KUKA KRL program: MyProgram_291().src

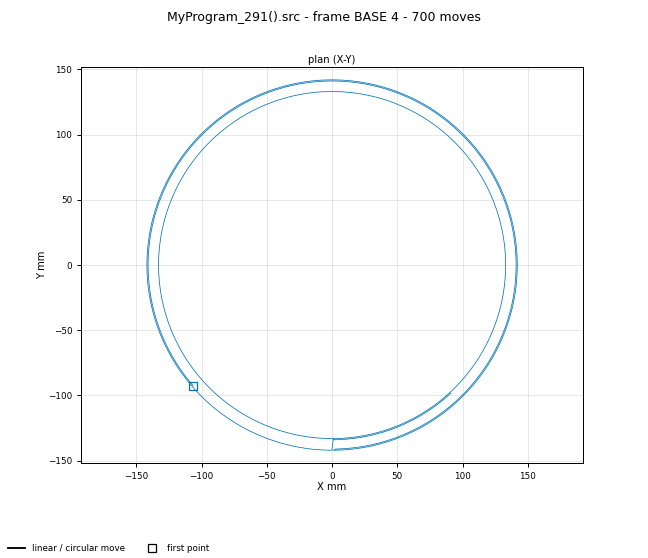
[picture p0: tool path of MyProgram_291().src in frame BASE 4, 700 of 700 moves have a stored position in this frame; points joined in program order, loops and branches not executed]
&ACCESS RVP
&REL 1
&PARAM TEMPLATE = C:\KRC\Roboter\Template\vorgabe
&PARAM EDITMASK = *
DEF MyProgram_291()
; ---- Setting reference (Base) ----
$BASE = BASE_DATA[4]

; --------------------------
; ---- Setting tool (TCP) ----
$TOOL = TOOL_DATA[3]
; --------------------------

$VEL.CP = VEL_APROX_PRINT
Startdeposition()
$VEL.CP = VEL_PRINT
LIN {X -106.5976,Y -92.4172,Z 176,A -136.4755,B 6.9518,C 0.3757,E1 6.8407,E2 228.6931} C_DIS
LIN {X -109.4772,Y -88.9868,Z 176,A -138.3075,B 6.952,C 0.3719,E1 6.8374,E2 230.5261} C_DIS
LIN {X -112.3182,Y -85.3731,Z 176,A -140.1975,B 6.9522,C 0.3681,E1 6.8342,E2 232.4184} C_DIS
LIN {X -114.9882,Y -81.7412,Z 176,A -142.0435,B 6.9524,C 0.3642,E1 6.8312,E2 234.2657} C_DIS
LIN {X -117.5398,Y -78.0276,Z 176,A -143.785,B 6.9527,C 0.3587,E1 6.8285,E2 235.9948} C_DIS
LIN {X -119.6611,Y -74.7331,Z 176,A -145.5405,B 6.9527,C 0.3571,E1 6.8258,E2 237.771} C_DIS
LIN {X -122.1664,Y -70.5632,Z 176,A -148.2334,B 6.9525,C 0.3616,E1 6.8219,E2 240.5556} C_DIS
LIN {X -125.0381,Y -65.3358,Z 176,A -149.8985,B 6.9533,C 0.3458,E1 6.8199,E2 242.1216} C_DIS
LIN {X -126.4778,Y -62.5025,Z 176,A -151.2741,B 6.9534,C 0.3436,E1 6.8181,E2 243.5075} C_DIS
LIN {X -128.0398,Y -59.237,Z 176,A -152.7086,B 6.9536,C 0.3394,E1 6.8164,E2 244.9366} C_DIS
LIN {X -129.8391,Y -55.1885,Z 176,A -154.746,B 6.9537,C 0.3378,E1 6.8141,E2 247.0039} C_DIS
LIN {X -131.2968,Y -51.6206,Z 176,A -156.1181,B 6.954,C 0.3312,E1 6.8127,E2 248.35} C_DIS
LIN {X -132.5485,Y -48.3154,Z 176,A -157.6493,B 6.9541,C 0.3286,E1 6.8112,E2 249.8927} C_DIS
LIN {X -133.6813,Y -45.0871,Z 176,A -158.9184,B 6.9544,C 0.3233,E1 6.8101,E2 251.1454} C_DIS
LIN {X -134.8654,Y -41.4075,Z 176,A -160.6121,B 6.9545,C 0.3207,E1 6.8086,E2 252.854} C_DIS
LIN {X -135.8285,Y -38.13,Z 176,A -162.047,B 6.9547,C 0.3175,E1 6.8075,E2 254.2942} C_DIS
LIN {X -136.7359,Y -34.7357,Z 176,A -163.3925,B 6.9549,C 0.3125,E1 6.8066,E2 255.628} C_DIS
LIN {X -137.4207,Y -31.9236,Z 176,A -164.649,B 6.9549,C 0.3103,E1 6.8058,E2 256.8943} C_DIS
LIN {X -138.1072,Y -28.8125,Z 176,A -165.9668,B 6.9551,C 0.307,E1 6.805,E2 258.2142} C_DIS
LIN {X -138.843,Y -25.0187,Z 176,A -167.6355,B 6.9553,C 0.3038,E1 6.8041,E2 259.8946} C_DIS
LIN {X -139.8868,Y -18.3035,Z 176,A -170.3898,B 6.9556,C 0.2959,E1 6.803,E2 262.6461} C_DIS
LIN {X -140.6363,Y -11.191,Z 176,A -173.5234,B 6.9558,C 0.2905,E1 6.8021,E2 265.8071} C_DIS
LIN {X -140.8895,Y -7.3194,Z 176,A -175.0544,B 6.956,C 0.2855,E1 6.8018,E2 267.3309} C_DIS
LIN {X -141.0677,Y -1.8699,Z 176,A -177.6099,B 6.9561,C 0.2833,E1 6.8017,E2 269.9283} C_DIS
LIN {X -141.0709,Y 1.6738,Z 176,A -178.7902,B 6.9564,C 0.276,E1 6.8017,E2 271.0743} C_DIS
LIN {X -140.9646,Y 5.6916,Z 176,A 179.5595,B 6.9566,C 0.2715,E1 6.8019,E2 272.7255} C_DIS
LIN {X -140.7276,Y 9.9587,Z 176,A 177.6568,B 6.9567,C 0.2686,E1 6.8022,E2 274.6481} C_DIS
LIN {X -139.9779,Y 17.6081,Z 176,A 174.5631,B 6.9571,C 0.2594,E1 6.8031,E2 277.7356} C_DIS
LIN {X -139.1333,Y 23.3505,Z 176,A 172.4063,B 6.9574,C 0.2502,E1 6.804,E2 279.8646} C_DIS
LIN {X -138.0178,Y 29.235,Z 176,A 169.7084,B 6.9575,C 0.2466,E1 6.8054,E2 282.5944} C_DIS
LIN {X -137.2534,Y 32.6338,Z 176,A 168.2329,B 6.9576,C 0.2434,E1 6.8064,E2 284.0764} C_DIS
LIN {X -136.4401,Y 35.8831,Z 176,A 166.9723,B 6.9578,C 0.2384,E1 6.8072,E2 285.3229} C_DIS
LIN {X -135.6663,Y 38.71,Z 176,A 165.682,B 6.9578,C 0.2363,E1 6.8082,E2 286.625} C_DIS
LIN {X -134.5047,Y 42.5661,Z 176,A 163.9944,B 6.958,C 0.2325,E1 6.8096,E2 288.3177} C_DIS
LIN {X -133.4991,Y 45.6249,Z 176,A 162.7591,B 6.9582,C 0.228,E1 6.8107,E2 289.5425} C_DIS
LIN {X -132.5325,Y 48.3598,Z 176,A 161.3126,B 6.9582,C 0.2282,E1 6.8121,E2 291.0221} C_DIS
LIN {X -130.963,Y 52.4595,Z 176,A 159.6682,B 6.9584,C 0.2216,E1 6.8137,E2 292.6472} C_DIS
LIN {X -129.7507,Y 55.3932,Z 176,A 158.4153,B 6.9584,C 0.2178,E1 6.8151,E2 293.8943} C_DIS
LIN {X -126.7522,Y 61.9464,Z 176,A 155.2826,B 6.9586,C 0.2127,E1 6.8188,E2 297.0504} C_DIS
LIN {X -124.96,Y 65.4845,Z 176,A 153.768,B 6.9588,C 0.2074,E1 6.8207,E2 298.5513} C_DIS
LIN {X -123.1422,Y 68.8468,Z 176,A 151.9508,B 6.9588,C 0.2068,E1 6.8232,E2 300.4007} C_DIS
LIN {X -120.7309,Y 72.9919,Z 176,A 150.2385,B 6.959,C 0.199,E1 6.8256,E2 302.0813} C_DIS
LIN {X -118.0913,Y 77.1907,Z 176,A 147.9543,B 6.959,C 0.1976,E1 6.8291,E2 304.3979} C_DIS
LIN {X -115.4613,Y 81.0712,Z 176,A 146.0801,B 6.9592,C 0.1927,E1 6.832,E2 306.2666} C_DIS
LIN {X -113.0544,Y 84.3949,Z 176,A 144.0965,B 6.9592,C 0.1929,E1 6.8354,E2 308.2885} C_DIS
LIN {X -110.7907,Y 87.3456,Z 176,A 142.9101,B 6.9594,C 0.1853,E1 6.8374,E2 309.4328} C_DIS
LIN {X -108.0272,Y 90.7409,Z 176,A 140.8316,B 6.9594,C 0.1852,E1 6.8411,E2 311.5475} C_DIS
LIN {X -105.8735,Y 93.245,Z 176,A 139.775,B 6.9596,C 0.1786,E1 6.843,E2 312.5669} C_DIS
LIN {X -101.406,Y 98.0847,Z 176,A 136.9788,B 6.9596,C 0.1746,E1 6.8484,E2 315.3761} C_DIS
LIN {X -98.5723,Y 100.9324,Z 176,A 135.3459,B 6.9598,C 0.1713,E1 6.8516,E2 317.0077} C_DIS
LIN {X -96.2529,Y 103.1464,Z 176,A 133.8537,B 6.9598,C 0.1713,E1 6.8547,E2 318.5226} C_DIS
LIN {X -90.6149,Y 108.1329,Z 176,A 130.9082,B 6.9599,C 0.164,E1 6.8609,E2 321.4514} C_DIS
LIN {X -88.1633,Y 110.1415,Z 176,A 129.2953,B 6.9599,C 0.166,E1 6.8645,E2 323.1043} C_DIS
LIN {X -85.2596,Y 112.404,Z 176,A 127.5101,B 6.9599,C 0.1673,E1 6.8685,E2 324.9244} C_DIS
LIN {X -81.0831,Y 115.453,Z 176,A 125.9883,B 6.9601,C 0.156,E1 6.8718,E2 326.372} C_DIS
LIN {X -78.3953,Y 117.2943,Z 176,A 124.5912,B 6.9601,C 0.1549,E1 6.8751,E2 327.7773} C_DIS
LIN {X -74.9843,Y 119.5043,Z 176,A 122.8795,B 6.9601,C 0.1532,E1 6.8791,E2 329.4954} C_DIS
LIN {X -71.4097,Y 121.6735,Z 176,A 121.401,B 6.9603,C 0.1477,E1 6.8826,E2 330.9448} C_DIS
LIN {X -68.0175,Y 123.6023,Z 176,A 119.6764,B 6.9603,C 0.1474,E1 6.8868,E2 332.6858} C_DIS
LIN {X -64.4592,Y 125.4929,Z 176,A 117.9731,B 6.9603,C 0.1461,E1 6.891,E2 334.3962} C_DIS
LIN {X -61.4649,Y 126.9874,Z 176,A 116.3879,B 6.9603,C 0.1476,E1 6.8951,E2 336.0088} C_DIS
LIN {X -58.5094,Y 128.3762,Z 176,A 115.1596,B 6.9603,C 0.1446,E1 6.8982,E2 337.2238} C_DIS
LIN {X -54.9539,Y 129.9373,Z 176,A 113.6452,B 6.9604,C 0.142,E1 6.902,E2 338.7292} C_DIS
LIN {X -52.0455,Y 131.1299,Z 176,A 112.3163,B 6.9604,C 0.1414,E1 6.9055,E2 340.0638} C_DIS
LIN {X -47.7422,Y 132.7552,Z 176,A 110.4599,B 6.9604,C 0.1393,E1 6.9104,E2 341.9174} C_DIS
LIN {X -43.7461,Y 134.1277,Z 176,A 108.659,B 6.9604,C 0.139,E1 6.9152,E2 343.7278} C_DIS
LIN {X -39.3613,Y 135.477,Z 176,A 106.9855,B 6.9606,C 0.1348,E1 6.9196,E2 345.3762} C_DIS
LIN {X -36.4098,Y 136.2996,Z 176,A 105.283,B 6.9605,C 0.1405,E1 6.9243,E2 347.1352} C_DIS
LIN {X -32.2916,Y 137.3359,Z 176,A 103.1946,B 6.9604,C 0.1446,E1 6.9301,E2 349.268} C_DIS
LIN {X -26.4655,Y 138.5744,Z 176,A 101.1582,B 6.9605,C 0.1377,E1 6.9356,E2 351.2552} C_DIS
LIN {X -22.5704,Y 139.2628,Z 176,A 99.7232,B 6.9605,C 0.1345,E1 6.9395,E2 352.6679} C_DIS
LIN {X -17.6999,Y 139.9659,Z 176,A 97.811,B 6.9606,C 0.1325,E1 6.9447,E2 354.5682} C_DIS
LIN {X -12.7549,Y 140.5032,Z 176,A 95.7582,B 6.9606,C 0.1324,E1 6.9504,E2 356.624} C_DIS
LIN {X -9.1693,Y 140.7818,Z 176,A 94.5714,B 6.9606,C 0.128,E1 6.9536,E2 357.7755} C_DIS
LIN {X -5.7888,Y 140.9608,Z 176,A 92.9782,B 6.9606,C 0.1311,E1 6.9582,E2 359.3957} C_DIS
LIN {X -2.2272,Y 141.0618,Z 176,A 91.6222,B 6.9606,C 0.1296,E1 6.9619,E2 360.7395} C_DIS
LIN {X 1.9978,Y 141.0656,Z 176,A 89.8711,B 6.9606,C 0.1302,E1 6.9668,E2 362.4943} C_DIS
LIN {X 5.9524,Y 140.9544,Z 176,A 88.2159,B 6.9606,C 0.1311,E1 6.9714,E2 364.1549} C_DIS
LIN {X 10.3005,Y 140.7027,Z 176,A 86.6003,B 6.9606,C 0.1291,E1 6.9759,E2 365.7505} C_DIS
LIN {X 13.1854,Y 140.462,Z 176,A 85.4424,B 6.9606,C 0.1291,E1 6.9791,E2 366.9057} C_DIS
LIN {X 15.9925,Y 140.1716,Z 176,A 84.1993,B 6.9606,C 0.131,E1 6.9826,E2 368.1607} C_DIS
LIN {X 19.9883,Y 139.6559,Z 176,A 82.5775,B 6.9606,C 0.1314,E1 6.9871,E2 369.7801} C_DIS
LIN {X 24.0859,Y 139.01,Z 176,A 80.9387,B 6.9606,C 0.1315,E1 6.9916,E2 371.4127} C_DIS
LIN {X 27.7172,Y 138.3301,Z 176,A 79.5231,B 6.9606,C 0.131,E1 6.9954,E2 372.8171} C_DIS
LIN {X 31.6691,Y 137.4788,Z 176,A 77.75,B 6.9606,C 0.1341,E1 7.0003,E2 374.6064} C_DIS
LIN {X 37.2187,Y 136.0834,Z 176,A 75.4221,B 6.9606,C 0.1359,E1 7.0066,E2 376.9343} C_DIS
LIN {X 40.2573,Y 135.2147,Z 176,A 74.196,B 6.9606,C 0.1359,E1 7.0099,E2 378.1529} C_DIS
LIN {X 44.1722,Y 133.986,Z 176,A 72.4661,B 6.9605,C 0.1385,E1 7.0145,E2 379.8905} C_DIS
LIN {X 47.3554,Y 132.8946,Z 176,A 71.1565,B 6.9605,C 0.1389,E1 7.0179,E2 381.1927} C_DIS
LIN {X 51.1487,Y 131.4802,Z 176,A 69.5776,B 6.9605,C 0.1395,E1 7.022,E2 382.763} C_DIS
LIN {X 53.7567,Y 130.4373,Z 176,A 68.3409,B 6.9605,C 0.1423,E1 7.0253,E2 384.0118} C_DIS
LIN {X 57.7524,Y 128.7163,Z 176,A 66.6133,B 6.9604,C 0.1437,E1 7.0297,E2 385.7342} C_DIS
LIN {X 61.749,Y 126.8496,Z 176,A 64.7824,B 6.9604,C 0.1466,E1 7.0343,E2 387.5702} C_DIS
LIN {X 67.1197,Y 124.0922,Z 176,A 62.3384,B 6.9603,C 0.1497,E1 7.0403,E2 390.0132} C_DIS
LIN {X 71.213,Y 121.789,Z 176,A 60.4497,B 6.9603,C 0.1521,E1 7.0449,E2 391.8996} C_DIS
LIN {X 74.9282,Y 119.5397,Z 176,A 58.7742,B 6.9602,C 0.1533,E1 7.0489,E2 393.564} C_DIS
LIN {X 78.2792,Y 117.3718,Z 176,A 57.3123,B 6.9602,C 0.1531,E1 7.0522,E2 395.0057} C_DIS
LIN {X 81.4199,Y 115.2154,Z 176,A 55.5916,B 6.9601,C 0.1586,E1 7.0562,E2 396.7487} C_DIS
LIN {X 85.2388,Y 112.4198,Z 176,A 53.6799,B 6.9601,C 0.1617,E1 7.0605,E2 398.6594} C_DIS
LIN {X 88.9491,Y 109.508,Z 176,A 51.7826,B 6.9599,C 0.1648,E1 7.0646,E2 400.5546} C_DIS
LIN {X 92.6938,Y 106.3562,Z 176,A 50.0338,B 6.9599,C 0.1643,E1 7.0683,E2 402.2733} C_DIS
LIN {X 99.2583,Y 100.2578,Z 176,A 46.2547,B 6.9597,C 0.174,E1 7.076,E2 406.0714} C_DIS
LIN {X 102.4648,Y 96.9783,Z 176,A 44.4276,B 6.9597,C 0.1772,E1 7.0796,E2 407.8945} C_DIS
LIN {X 104.8841,Y 94.3568,Z 176,A 42.9712,B 6.9595,C 0.1804,E1 7.0823,E2 409.3523} C_DIS
LIN {X 107.6922,Y 91.1386,Z 176,A 40.3692,B 6.959,C 0.1996,E1 7.0872,E2 412.0647} C_DIS
LIN {X 112.3745,Y 85.2989,Z 176,A 38.269,B 6.9593,C 0.1897,E1 7.0906,E2 414.0472} C_DIS
LIN {X 115.159,Y 81.4998,Z 176,A 36.5374,B 6.9593,C 0.1908,E1 7.0934,E2 415.7564} C_DIS
LIN {X 117.3119,Y 78.369,Z 176,A 34.9703,B 6.9592,C 0.1949,E1 7.0958,E2 417.3272} C_DIS
LIN {X 119.4142,Y 75.127,Z 176,A 33.4308,B 6.9591,C 0.1982,E1 7.0981,E2 418.8636} C_DIS
LIN {X 121.432,Y 71.8206,Z 176,A 31.9579,B 6.9591,C 0.2002,E1 7.1002,E2 420.3244} C_DIS
LIN {X 123.5711,Y 68.074,Z 176,A 30.1098,B 6.9588,C 0.2063,E1 7.1028,E2 422.1857} C_DIS
LIN {X 125.5535,Y 64.3403,Z 176,A 28.5885,B 6.9588,C 0.2071,E1 7.1047,E2 423.6827} C_DIS
LIN {X 127.281,Y 60.8503,Z 176,A 27.0023,B 6.9587,C 0.2112,E1 7.1067,E2 425.2703} C_DIS
LIN {X 128.5679,Y 58.0842,Z 176,A 25.8251,B 6.9587,C 0.2133,E1 7.108,E2 426.4403} C_DIS
LIN {X 130.0336,Y 54.7232,Z 176,A 24.0309,B 6.9583,C 0.2228,E1 7.1101,E2 428.2747} C_DIS
LIN {X 131.2459,Y 51.7515,Z 176,A 22.8885,B 6.9583,C 0.2233,E1 7.1112,E2 429.3972} C_DIS
LIN {X 132.5413,Y 48.3353,Z 176,A 21.5624,B 6.9583,C 0.2244,E1 7.1125,E2 430.7039} C_DIS
LIN {X 133.6036,Y 45.3205,Z 176,A 20.2936,B 6.9582,C 0.2274,E1 7.1136,E2 431.9698} C_DIS
LIN {X 134.8252,Y 41.5389,Z 176,A 18.6838,B 6.958,C 0.2317,E1 7.115,E2 433.58} C_DIS
LIN {X 135.8092,Y 38.1992,Z 176,A 17.3473,B 6.958,C 0.2341,E1 7.116,E2 434.9075} C_DIS
LIN {X 136.9729,Y 33.7976,Z 176,A 15.3871,B 6.9577,C 0.2413,E1 7.1174,E2 436.8834} C_DIS
LIN {X 137.737,Y 30.5352,Z 176,A 14.1817,B 6.9577,C 0.2422,E1 7.1181,E2 438.0697} C_DIS
LIN {X 138.5004,Y 26.8529,Z 176,A 12.829,B 6.9577,C 0.2432,E1 7.1189,E2 439.4008} C_DIS
LIN {X 139.1219,Y 23.4186,Z 176,A 11.4105,B 6.9575,C 0.2472,E1 7.1196,E2 440.8205} C_DIS
LIN {X 139.5094,Y 20.9948,Z 176,A 10.1393,B 6.9572,C 0.2552,E1 7.1201,E2 442.1281} C_DIS
LIN {X 140.1341,Y 16.3069,Z 176,A 8.439,B 6.9572,C 0.2565,E1 7.1207,E2 443.8013} C_DIS
LIN {X 140.4477,Y 13.3341,Z 176,A 7.2773,B 6.9571,C 0.259,E1 7.121,E2 444.9572} C_DIS
LIN {X 140.7204,Y 10.0574,Z 176,A 5.8794,B 6.9569,C 0.264,E1 7.1213,E2 446.3642} C_DIS
LIN {X 140.9315,Y 6.4829,Z 176,A 4.3562,B 6.9567,C 0.2695,E1 7.1216,E2 447.8976} C_DIS
LIN {X 141.0606,Y 2.2991,Z 176,A 2.9218,B 6.9567,C 0.2694,E1 7.1216,E2 449.2988} C_DIS
LIN {X 141.0755,Y -1.1811,Z 176,A 1.2595,B 6.9563,C 0.2781,E1 7.1216,E2 450.9947} C_DIS
LIN {X 140.9888,Y -5.0699,Z 176,A 0.0079,B 6.9564,C 0.2765,E1 7.1216,E2 452.205} C_DIS
LIN {X 140.8658,Y -7.7902,Z 176,A -1.2897,B 6.9561,C 0.2833,E1 7.1214,E2 453.5285} C_DIS
LIN {X 140.5898,Y -11.7421,Z 176,A -2.6938,B 6.9561,C 0.284,E1 7.1211,E2 454.9073} C_DIS
LIN {X 140.3246,Y -14.5812,Z 176,A -3.7947,B 6.9561,C 0.2862,E1 7.1208,E2 456.0018} C_DIS
LIN {X 139.9717,Y -17.6551,Z 176,A -5.2781,B 6.9557,C 0.2941,E1 7.1203,E2 457.5159} C_DIS
LIN {X 139.4569,Y -21.3344,Z 176,A -6.4972,B 6.9557,C 0.2929,E1 7.1198,E2 458.6985} C_DIS
LIN {X 138.9672,Y -24.3247,Z 176,A -7.9014,B 6.9554,C 0.2997,E1 7.1191,E2 460.1265} C_DIS
LIN {X 138.0027,Y -29.3047,Z 176,A -9.8882,B 6.9553,C 0.3042,E1 7.118,E2 462.1056} C_DIS
LIN {X 137.0687,Y -33.4003,Z 176,A -11.5987,B 6.955,C 0.3091,E1 7.1169,E2 463.8183} C_DIS
LIN {X 134.9357,Y -41.1779,Z 176,A -14.7519,B 6.9547,C 0.3159,E1 7.1146,E2 466.9585} C_DIS
LIN {X 133.8895,Y -44.4619,Z 176,A -16.0341,B 6.9547,C 0.3175,E1 7.1135,E2 468.2266} C_DIS
LIN {X 132.259,Y -49.1014,Z 176,A -17.9439,B 6.9545,C 0.3213,E1 7.1117,E2 470.1269} C_DIS
LIN {X 131.0152,Y -52.3302,Z 176,A -19.4921,B 6.9542,C 0.3278,E1 7.1101,E2 471.6952} C_DIS
LIN {X 129.8222,Y -55.2277,Z 176,A -20.715,B 6.9541,C 0.3303,E1 7.1088,E2 472.9129} C_DIS
LIN {X 128.5523,Y -58.1192,Z 176,A -21.9622,B 6.9539,C 0.333,E1 7.1074,E2 474.1566} C_DIS
LIN {X 127.272,Y -60.8691,Z 176,A -23.8015,B 6.9532,C 0.3476,E1 7.1051,E2 476.0766} C_DIS
LIN {X 124.8146,Y -65.7613,Z 176,A -25.2594,B 6.9536,C 0.3391,E1 7.1033,E2 477.4364} C_DIS
LIN {X 122.8185,Y -69.4227,Z 176,A -27.0945,B 6.9533,C 0.3461,E1 7.1008,E2 479.2919} C_DIS
LIN {X 120.9907,Y -72.5614,Z 176,A -28.9213,B 6.9528,C 0.3563,E1 7.0981,E2 481.1662} C_DIS
LIN {X 118.6271,Y -76.3643,Z 176,A -30.3307,B 6.9529,C 0.3533,E1 7.0961,E2 482.5237} C_DIS
LIN {X 116.15,Y -80.0815,Z 176,A -32.0828,B 6.9528,C 0.3565,E1 7.0933,E2 484.2694} C_DIS
LIN {X 114.2154,Y -82.8167,Z 176,A -33.7708,B 6.9523,C 0.3658,E1 7.0905,E2 486.0017} C_DIS
LIN {X 111.7275,Y -86.1436,Z 176,A -35.1944,B 6.9523,C 0.3649,E1 7.0881,E2 487.3923} C_DIS
LIN {X 108.7402,Y -89.8852,Z 176,A -36.9542,B 6.9523,C 0.3659,E1 7.0851,E2 489.1297} C_DIS
LIN {X 106.1955,Y -92.8779,Z 176,A -38.5271,B 6.9521,C 0.3691,E1 7.0822,E2 490.7011} C_DIS
LIN {X 103.8823,Y -95.458,Z 176,A -39.8642,B 6.9521,C 0.3709,E1 7.0797,E2 492.0303} C_DIS
LIN {X 101.2064,Y -98.2908,Z 176,A -41.4737,B 6.9518,C 0.3748,E1 7.0766,E2 493.6448} C_DIS
LIN {X 98.3144,Y -101.1836,Z 176,A -43.139,B 6.9516,C 0.3783,E1 7.0733,E2 495.3121} C_DIS
LIN {X 95.2304,Y -104.0916,Z 176,A -44.8391,B 6.9515,C 0.3814,E1 7.0698,E2 497.011} C_DIS
LIN {X 92.663,Y -106.3831,Z 176,A -46.2184,B 6.9513,C 0.3839,E1 7.0669,E2 498.3892} C_DIS
LIN {X 89.4376,Y -109.1088,Z 176,A -47.8775,B 6.9513,C 0.3862,E1 7.0634,E2 500.0425} C_DIS
LIN {X 86.3647,Y -111.5568,Z 176,A -49.4568,B 6.9511,C 0.3888,E1 7.0599,E2 501.621} C_DIS
LIN {X 82.88,Y -114.1696,Z 176,A -51.1295,B 6.951,C 0.3903,E1 7.0562,E2 503.2826} C_DIS
LIN {X 78.9966,Y -116.8902,Z 176,A -53.1182,B 6.9507,C 0.3947,E1 7.0516,E2 505.2813} C_DIS
LIN {X 75.2872,Y -119.3131,Z 176,A -54.8838,B 6.9506,C 0.3971,E1 7.0474,E2 507.0439} C_DIS
LIN {X 72.528,Y -121.0107,Z 176,A -56.6461,B 6.95,C 0.407,E1 7.0431,E2 508.8662} C_DIS
LIN {X 68.522,Y -123.3229,Z 176,A -58.0988,B 6.9503,C 0.4024,E1 7.0397,E2 510.2644} C_DIS
LIN {X 64.3361,Y -125.5556,Z 176,A -60.0871,B 6.9501,C 0.4062,E1 7.0347,E2 512.2623} C_DIS
LIN {X 59.8205,Y -127.77,Z 176,A -61.8483,B 6.9501,C 0.4041,E1 7.0304,E2 513.9879} C_DIS
LIN {X 55.231,Y -129.8208,Z 176,A -63.9394,B 6.95,C 0.4075,E1 7.025,E2 516.0872} C_DIS
LIN {X 51.8202,Y -131.2192,Z 176,A -65.4654,B 6.9499,C 0.4098,E1 7.021,E2 517.6182} C_DIS
LIN {X 48.779,Y -132.3798,Z 176,A -66.8136,B 6.9497,C 0.4117,E1 7.0175,E2 518.9708} C_DIS
LIN {X 44.8676,Y -133.7544,Z 176,A -68.5597,B 6.9496,C 0.4145,E1 7.0129,E2 520.7263} C_DIS
LIN {X 40.5679,Y -135.1224,Z 176,A -70.3527,B 6.9496,C 0.4156,E1 7.0081,E2 522.5154} C_DIS
LIN {X 35.6572,Y -136.5004,Z 176,A -72.33,B 6.9496,C 0.4158,E1 7.0028,E2 524.4817} C_DIS
LIN {X 31.6081,Y -137.4927,Z 176,A -73.9074,B 6.9496,C 0.4152,E1 6.9985,E2 526.0448} C_DIS
LIN {X 28.272,Y -138.2172,Z 176,A -75.168,B 6.9496,C 0.414,E1 6.9951,E2 527.2895} C_DIS
LIN {X 24.9732,Y -138.8512,Z 176,A -76.7201,B 6.9494,C 0.4181,E1 6.9908,E2 528.8675} C_DIS
LIN {X 20.7766,Y -139.543,Z 176,A -78.6261,B 6.9491,C 0.422,E1 6.9855,E2 530.7982} C_DIS
LIN {X 16.7485,Y -140.0815,Z 176,A -80.0165,B 6.9493,C 0.4185,E1 6.9817,E2 532.1551} C_DIS
LIN {X 13.7667,Y -140.4062,Z 176,A -81.215,B 6.9493,C 0.4187,E1 6.9784,E2 533.3517} C_DIS
LIN {X 10.7106,Y -140.6728,Z 176,A -82.3844,B 6.9493,C 0.4179,E1 6.9752,E2 534.5115} C_DIS
LIN {X 7.4209,Y -140.8844,Z 176,A -83.9743,B 6.9491,C 0.4224,E1 6.9706,E2 536.1355} C_DIS
LIN {X 2.6587,Y -141.0546,Z 176,A -85.7031,B 6.9493,C 0.4194,E1 6.9659,E2 537.8379} C_DIS
LIN {X 2.6587,Y -141.0546,Z 176,A -85.7031,B 6.9493,C 0.4194,E1 6.9659,E2 537.8379} C_DIS
Enddeposition()
LIN {X 1.0477,Y -141.9797,Z 176,A -86.1978,B 6.9491,C 0.4209,E1 6.9643,E2 538.3447} C_DIS
Startdeposition()
$VEL.CP = VEL_PRINT
LIN {X 3.343,Y -141.9469,Z 176,A -84.8295,B 6.9495,C 0.4135,E1 6.9683,E2 536.9165} C_DIS
LIN {X 6.7269,Y -141.8261,Z 176,A -83.4813,B 6.9495,C 0.4135,E1 6.9721,E2 535.5701} C_DIS
LIN {X 9.9965,Y -141.633,Z 176,A -82.1304,B 6.9495,C 0.4126,E1 6.9759,E2 534.2145} C_DIS
LIN {X 13.7808,Y -141.3147,Z 176,A -80.6591,B 6.9495,C 0.413,E1 6.9799,E2 532.7506} C_DIS
LIN {X 17.3767,Y -140.9186,Z 176,A -79.2242,B 6.9495,C 0.4128,E1 6.9839,E2 531.3183} C_DIS
LIN {X 20.8496,Y -140.4478,Z 176,A -77.8083,B 6.9495,C 0.412,E1 6.9878,E2 529.9014} C_DIS
LIN {X 24.2877,Y -139.894,Z 176,A -76.4424,B 6.9495,C 0.4119,E1 6.9916,E2 528.54} C_DIS
LIN {X 27.5706,Y -139.2842,Z 176,A -75.0559,B 6.9497,C 0.4103,E1 6.9954,E2 527.1473} C_DIS
LIN {X 30.5505,Y -138.6603,Z 176,A -73.7316,B 6.9498,C 0.4078,E1 6.999,E2 525.8092} C_DIS
LIN {X 34.487,Y -137.7334,Z 176,A -72.2551,B 6.9498,C 0.4092,E1 7.003,E2 524.3527} C_DIS
LIN {X 37.7193,Y -136.8838,Z 176,A -70.995,B 6.9498,C 0.4095,E1 7.0064,E2 523.1037} C_DIS
LIN {X 41.2128,Y -135.8722,Z 176,A -69.4805,B 6.9498,C 0.4074,E1 7.0104,E2 521.5819} C_DIS
LIN {X 44.42,Y -134.858,Z 176,A -68.2173,B 6.9498,C 0.4076,E1 7.0138,E2 520.3303} C_DIS
LIN {X 47.7142,Y -133.728,Z 176,A -66.6798,B 6.9501,C 0.4039,E1 7.0179,E2 518.774} C_DIS
LIN {X 50.9768,Y -132.5187,Z 176,A -65.2879,B 6.9501,C 0.4025,E1 7.0215,E2 517.3828} C_DIS
LIN {X 54.3352,Y -131.1771,Z 176,A -63.8014,B 6.9503,C 0.4003,E1 7.0254,E2 515.8915} C_DIS
LIN {X 58.2843,Y -129.4706,Z 176,A -62.1262,B 6.9503,C 0.3992,E1 7.0296,E2 514.2232} C_DIS
LIN {X 61.4279,Y -128.0088,Z 176,A -60.7317,B 6.9504,C 0.3974,E1 7.0332,E2 512.8282} C_DIS
LIN {X 64.5346,Y -126.4709,Z 176,A -59.3333,B 6.9505,C 0.3954,E1 7.0366,E2 511.4287} C_DIS
LIN {X 67.6372,Y -124.842,Z 176,A -57.9121,B 6.9507,C 0.3933,E1 7.0402,E2 510.0054} C_DIS
LIN {X 71.4568,Y -122.6956,Z 176,A -56.1815,B 6.9507,C 0.3913,E1 7.0443,E2 508.2784} C_DIS
LIN {X 75.1782,Y -120.4509,Z 176,A -54.4454,B 6.9509,C 0.3888,E1 7.0485,E2 506.5433} C_DIS
LIN {X 78.8259,Y -118.0959,Z 176,A -52.724,B 6.951,C 0.3864,E1 7.0525,E2 504.8245} C_DIS
LIN {X 81.7121,Y -116.1176,Z 176,A -51.3441,B 6.9511,C 0.3846,E1 7.0556,E2 503.4477} C_DIS
LIN {X 84.5343,Y -114.0798,Z 176,A -49.9434,B 6.9513,C 0.3821,E1 7.0588,E2 502.0464} C_DIS
LIN {X 87.3046,Y -111.9742,Z 176,A -48.5479,B 6.9514,C 0.3797,E1 7.0619,E2 500.6507} C_DIS
LIN {X 90.6931,Y -109.2471,Z 176,A -46.7171,B 6.9517,C 0.375,E1 7.0659,E2 498.8081} C_DIS
LIN {X 94.0114,Y -106.4049,Z 176,A -45.1007,B 6.9517,C 0.3742,E1 7.0692,E2 497.2099} C_DIS
LIN {X 96.5912,Y -104.0689,Z 176,A -43.6891,B 6.9519,C 0.3713,E1 7.0721,E2 495.7961} C_DIS
LIN {X 99.7343,Y -101.0614,Z 176,A -41.9709,B 6.952,C 0.3683,E1 7.0756,E2 494.0813} C_DIS
LIN {X 102.1809,Y -98.5863,Z 176,A -40.5778,B 6.9522,C 0.3655,E1 7.0783,E2 492.6884} C_DIS
LIN {X 105.1672,Y -95.394,Z 176,A -38.8536,B 6.9523,C 0.3624,E1 7.0816,E2 490.9679} C_DIS
LIN {X 107.518,Y -92.7364,Z 176,A -37.4597,B 6.9525,C 0.3599,E1 7.0841,E2 489.5777} C_DIS
LIN {X 109.7579,Y -90.0747,Z 176,A -35.9823,B 6.9527,C 0.3554,E1 7.0868,E2 488.0891} C_DIS
LIN {X 112.4882,Y -86.6415,Z 176,A -34.3351,B 6.9527,C 0.3536,E1 7.0896,E2 486.4568} C_DIS
LIN {X 114.5779,Y -83.8577,Z 176,A -32.942,B 6.9529,C 0.3505,E1 7.0919,E2 485.0639} C_DIS
LIN {X 117.0479,Y -80.3737,Z 176,A -31.2374,B 6.9531,C 0.3467,E1 7.0946,E2 483.3601} C_DIS
LIN {X 119.4479,Y -76.7621,Z 176,A -29.5307,B 6.9533,C 0.3432,E1 7.0972,E2 481.6576} C_DIS
LIN {X 121.4708,Y -73.5187,Z 176,A -27.9446,B 6.9535,C 0.3385,E1 7.0995,E2 480.0641} C_DIS
LIN {X 123.505,Y -70.0485,Z 176,A -26.4281,B 6.9536,C 0.3364,E1 7.1016,E2 478.5604} C_DIS
LIN {X 125.221,Y -66.9324,Z 176,A -25.0042,B 6.9538,C 0.333,E1 7.1035,E2 477.1366} C_DIS
LIN {X 126.8387,Y -63.812,Z 176,A -23.6316,B 6.9539,C 0.3302,E1 7.1053,E2 475.7688} C_DIS
LIN {X 128.5932,Y -60.198,Z 176,A -21.9442,B 6.9542,C 0.3246,E1 7.1073,E2 474.071} C_DIS
LIN {X 130.4477,Y -56.0633,Z 176,A -20.271,B 6.9542,C 0.3227,E1 7.1092,E2 472.4167} C_DIS
LIN {X 131.7814,Y -52.8519,Z 176,A -18.8531,B 6.9545,C 0.3187,E1 7.1107,E2 470.9956} C_DIS
LIN {X 133.084,Y -49.4811,Z 176,A -17.4392,B 6.9546,C 0.3156,E1 7.1121,E2 469.5863} C_DIS
LIN {X 134.2559,Y -46.2068,Z 176,A -16.0618,B 6.9548,C 0.3122,E1 7.1133,E2 468.211} C_DIS
LIN {X 135.3541,Y -42.8837,Z 176,A -14.6955,B 6.9548,C 0.3092,E1 7.1145,E2 466.8495} C_DIS
LIN {X 136.3368,Y -39.6481,Z 176,A -13.3271,B 6.9551,C 0.3054,E1 7.1156,E2 465.4793} C_DIS
LIN {X 137.3033,Y -36.1613,Z 176,A -11.9137,B 6.9551,C 0.3022,E1 7.1166,E2 464.0708} C_DIS
LIN {X 138.1139,Y -32.9292,Z 176,A -10.5967,B 6.9553,C 0.2989,E1 7.1175,E2 462.7562} C_DIS
LIN {X 138.9062,Y -29.4114,Z 176,A -9.1739,B 6.9555,C 0.2954,E1 7.1183,E2 461.3364} C_DIS
LIN {X 139.5896,Y -25.9788,Z 176,A -7.7925,B 6.9556,C 0.292,E1 7.1191,E2 459.9579} C_DIS
LIN {X 140.1627,Y -22.6839,Z 176,A -6.4725,B 6.9558,C 0.2888,E1 7.1197,E2 458.6406} C_DIS
LIN {X 140.6772,Y -19.2421,Z 176,A -5.1102,B 6.9558,C 0.2856,E1 7.1202,E2 457.2826} C_DIS
LIN {X 141.1056,Y -15.7881,Z 176,A -3.6978,B 6.9561,C 0.2814,E1 7.1207,E2 455.8679} C_DIS
LIN {X 141.4608,Y -12.1905,Z 176,A -2.2764,B 6.9562,C 0.2779,E1 7.121,E2 454.4502} C_DIS
LIN {X 141.7182,Y -8.6992,Z 176,A -0.8997,B 6.9563,C 0.2746,E1 7.1213,E2 453.077} C_DIS
LIN {X 141.8838,Y -5.3614,Z 176,A 0.4169,B 6.9565,C 0.2713,E1 7.1215,E2 451.7635} C_DIS
LIN {X 141.9788,Y -1.5286,Z 176,A 1.8535,B 6.9565,C 0.269,E1 7.1215,E2 450.3403} C_DIS
LIN {X 141.9824,Y 1,Z 176,A 3.036,B 6.9568,C 0.2629,E1 7.1215,E2 449.1355} C_DIS
LIN {X 141.8887,Y 5.2367,Z 176,A 4.6218,B 6.9568,C 0.2604,E1 7.1214,E2 447.5647} C_DIS
LIN {X 141.7259,Y 8.5746,Z 176,A 5.76,B 6.9568,C 0.2606,E1 7.1212,E2 446.4533} C_DIS
LIN {X 141.4731,Y 12.0449,Z 176,A 7.3083,B 6.9571,C 0.2538,E1 7.1209,E2 444.8847} C_DIS
LIN {X 141.1226,Y 15.6303,Z 176,A 8.7288,B 6.9572,C 0.2503,E1 7.1205,E2 443.4675} C_DIS
LIN {X 140.6929,Y 19.1225,Z 176,A 10.1141,B 6.9574,C 0.2469,E1 7.12,E2 442.0857} C_DIS
LIN {X 140.1831,Y 22.5621,Z 176,A 11.4827,B 6.9574,C 0.2436,E1 7.1194,E2 440.7206} C_DIS
LIN {X 139.6134,Y 25.8542,Z 176,A 12.8318,B 6.9576,C 0.2398,E1 7.1187,E2 439.3704} C_DIS
LIN {X 138.9376,Y 29.2662,Z 176,A 14.2047,B 6.9577,C 0.2364,E1 7.118,E2 438.0006} C_DIS
LIN {X 138.1472,Y 32.7907,Z 176,A 15.6303,B 6.9578,C 0.233,E1 7.1171,E2 436.5781} C_DIS
LIN {X 137.3369,Y 36.0354,Z 176,A 16.8447,B 6.9578,C 0.2318,E1 7.1162,E2 435.3806} C_DIS
LIN {X 136.5408,Y 38.9459,Z 176,A 18.2843,B 6.9581,C 0.2242,E1 7.1151,E2 433.9109} C_DIS
LIN {X 135.3554,Y 42.8796,Z 176,A 19.7335,B 6.9581,C 0.2237,E1 7.1139,E2 432.4881} C_DIS
LIN {X 134.3081,Y 46.0561,Z 176,A 21.0925,B 6.9583,C 0.2198,E1 7.1127,E2 431.127} C_DIS
LIN {X 133.1381,Y 49.3366,Z 176,A 22.4698,B 6.9583,C 0.2166,E1 7.1114,E2 429.7525} C_DIS
LIN {X 132.1234,Y 51.9939,Z 176,A 23.7505,B 6.9585,C 0.211,E1 7.1101,E2 428.4536} C_DIS
LIN {X 130.4963,Y 55.9507,Z 176,A 25.2871,B 6.9585,C 0.21,E1 7.1085,E2 426.941} C_DIS
LIN {X 128.9485,Y 59.4297,Z 176,A 26.8777,B 6.9587,C 0.205,E1 7.1066,E2 425.3423} C_DIS
LIN {X 127.2514,Y 62.9817,Z 176,A 28.3631,B 6.9587,C 0.2029,E1 7.1048,E2 423.8696} C_DIS
LIN {X 125.6284,Y 66.1596,Z 176,A 29.6854,B 6.9588,C 0.2014,E1 7.1031,E2 422.5619} C_DIS
LIN {X 123.9279,Y 69.2974,Z 176,A 31.3127,B 6.959,C 0.1943,E1 7.1009,E2 420.9095} C_DIS
LIN {X 121.7475,Y 73.0608,Z 176,A 33.0496,B 6.9591,C 0.1903,E1 7.0984,E2 419.1741} C_DIS
LIN {X 119.4523,Y 76.7551,Z 176,A 34.7679,B 6.9592,C 0.1868,E1 7.0959,E2 417.4599} C_DIS
LIN {X 117.0846,Y 80.3202,Z 176,A 36.3969,B 6.9592,C 0.1845,E1 7.0934,E2 415.8429} C_DIS
LIN {X 114.6024,Y 83.8243,Z 176,A 38.1436,B 6.9594,C 0.1802,E1 7.0905,E2 414.0937} C_DIS
LIN {X 111.9347,Y 87.3554,Z 176,A 39.821,B 6.9594,C 0.1782,E1 7.0877,E2 412.4298} C_DIS
LIN {X 109.2158,Y 90.7309,Z 176,A 41.5162,B 6.9595,C 0.1753,E1 7.0847,E2 410.741} C_DIS
LIN {X 106.8814,Y 93.4694,Z 176,A 43.0712,B 6.9597,C 0.1703,E1 7.0818,E2 409.172} C_DIS
LIN {X 104.071,Y 96.589,Z 176,A 44.6245,B 6.9597,C 0.1692,E1 7.0789,E2 407.6366} C_DIS
LIN {X 101.6238,Y 99.1609,Z 176,A 46.1145,B 6.9597,C 0.1653,E1 7.076,E2 406.1388} C_DIS
LIN {X 98.5368,Y 102.2289,Z 176,A 47.7609,B 6.9598,C 0.1637,E1 7.0728,E2 404.5062} C_DIS
LIN {X 95.9596,Y 104.6515,Z 176,A 49.1741,B 6.9598,C 0.1612,E1 7.0699,E2 403.0945} C_DIS
LIN {X 92.7896,Y 107.4721,Z 176,A 50.6918,B 6.9598,C 0.1614,E1 7.0667,E2 401.6017} C_DIS
LIN {X 90.7438,Y 109.2052,Z 176,A 51.9152,B 6.96,C 0.1569,E1 7.0641,E2 400.3598} C_DIS
LIN {X 88.0385,Y 111.3982,Z 176,A 53.3098,B 6.96,C 0.1546,E1 7.061,E2 398.9663} C_DIS
LIN {X 84.9983,Y 113.7344,Z 176,A 54.9293,B 6.9601,C 0.1506,E1 7.0574,E2 397.3372} C_DIS
LIN {X 81.7595,Y 116.0842,Z 176,A 56.422,B 6.9601,C 0.1501,E1 7.0541,E2 395.8602} C_DIS
LIN {X 78.8786,Y 118.0607,Z 176,A 57.8227,B 6.9601,C 0.148,E1 7.0508,E2 394.4605} C_DIS
LIN {X 75.9045,Y 119.9945,Z 176,A 59.3597,B 6.9602,C 0.1439,E1 7.0472,E2 392.9098} C_DIS
LIN {X 72.1169,Y 122.3085,Z 176,A 61.122,B 6.9602,C 0.1418,E1 7.043,E2 391.151} C_DIS
LIN {X 68.5234,Y 124.3575,Z 176,A 62.6784,B 6.9602,C 0.1414,E1 7.0392,E2 389.6093} C_DIS
LIN {X 65.4317,Y 126.0106,Z 176,A 64.0752,B 6.9603,C 0.1398,E1 7.0358,E2 388.2148} C_DIS
LIN {X 62.2038,Y 127.6351,Z 176,A 65.6594,B 6.9604,C 0.1358,E1 7.0317,E2 386.6143} C_DIS
LIN {X 58.2687,Y 129.4776,Z 176,A 67.3659,B 6.9604,C 0.1345,E1 7.0274,E2 384.914} C_DIS
LIN {X 55.0092,Y 130.8957,Z 176,A 68.7786,B 6.9604,C 0.1332,E1 7.0238,E2 383.5042} C_DIS
LIN {X 51.1029,Y 132.4697,Z 176,A 70.3582,B 6.9604,C 0.1335,E1 7.0197,E2 381.9403} C_DIS
LIN {X 48.4302,Y 133.4699,Z 176,A 71.6107,B 6.9605,C 0.1306,E1 7.0164,E2 380.6749} C_DIS
LIN {X 44.5419,Y 134.8175,Z 176,A 73.1498,B 6.9605,C 0.1311,E1 7.0124,E2 379.1518} C_DIS
LIN {X 41.3535,Y 135.8291,Z 176,A 74.4908,B 6.9605,C 0.1301,E1 7.0088,E2 377.8122} C_DIS
LIN {X 38.3278,Y 136.7136,Z 176,A 75.7751,B 6.9605,C 0.1289,E1 7.0054,E2 376.5266} C_DIS
LIN {X 34.4837,Y 137.7343,Z 176,A 77.3367,B 6.9605,C 0.1285,E1 7.0012,E2 374.971} C_DIS
LIN {X 31.2971,Y 138.4928,Z 176,A 78.6839,B 6.9605,C 0.1272,E1 6.9975,E2 373.6208} C_DIS
LIN {X 27.6926,Y 139.2594,Z 176,A 80.1254,B 6.9605,C 0.1271,E1 6.9936,E2 372.1856} C_DIS
LIN {X 24.2741,Y 139.8964,Z 176,A 81.5329,B 6.9605,C 0.1263,E1 6.9897,E2 370.778} C_DIS
LIN {X 20.975,Y 140.429,Z 176,A 82.8879,B 6.9605,C 0.1256,E1 6.9859,E2 369.4226} C_DIS
LIN {X 17.5085,Y 140.9029,Z 176,A 84.3127,B 6.9606,C 0.1248,E1 6.982,E2 367.9965} C_DIS
LIN {X 14.0483,Y 141.289,Z 176,A 85.7425,B 6.9606,C 0.124,E1 6.978,E2 366.564} C_DIS
LIN {X 10.4444,Y 141.6003,Z 176,A 87.2963,B 6.9606,C 0.1221,E1 6.9737,E2 364.9987} C_DIS
LIN {X 5.3522,Y 141.8842,Z 176,A 89.206,B 6.9606,C 0.1242,E1 6.9684,E2 363.1089} C_DIS
LIN {X 1.7343,Y 141.9758,Z 176,A 90.6287,B 6.9606,C 0.1247,E1 6.9644,E2 361.6917} C_DIS
LIN {X -1.7459,Y 141.9756,Z 176,A 92.1299,B 6.9606,C 0.1232,E1 6.9602,E2 360.1788} C_DIS
LIN {X -6.1991,Y 141.8512,Z 176,A 94.0243,B 6.9606,C 0.1219,E1 6.9549,E2 358.2727} C_DIS
LIN {X -10.1337,Y 141.623,Z 176,A 95.5073,B 6.9606,C 0.1238,E1 6.9508,E2 356.8043} C_DIS
LIN {X -13.79,Y 141.3138,Z 176,A 96.9622,B 6.9606,C 0.1246,E1 6.9467,E2 355.3535} C_DIS
LIN {X -17.3838,Y 140.9178,Z 176,A 98.4046,B 6.9606,C 0.1253,E1 6.9428,E2 353.9141} C_DIS
LIN {X -20.8312,Y 140.4504,Z 176,A 99.8289,B 6.9606,C 0.1255,E1 6.9388,E2 352.4879} C_DIS
LIN {X -24.3222,Y 139.8878,Z 176,A 101.2152,B 6.9606,C 0.1268,E1 6.935,E2 351.1076} C_DIS
LIN {X -27.5948,Y 139.2793,Z 176,A 102.6108,B 6.9606,C 0.1268,E1 6.9312,E2 349.7061} C_DIS
LIN {X -30.987,Y 138.5636,Z 176,A 104.0507,B 6.9606,C 0.127,E1 6.9272,E2 348.2618} C_DIS
LIN {X -34.4844,Y 137.7341,Z 176,A 105.3188,B 6.9606,C 0.1307,E1 6.9238,E2 347.018} C_DIS
LIN {X -37.7395,Y 136.8782,Z 176,A 106.8353,B 6.9606,C 0.1293,E1 6.9197,E2 345.4821} C_DIS
LIN {X -41.2158,Y 135.8713,Z 176,A 108.3032,B 6.9606,C 0.1304,E1 6.9158,E2 344.0142} C_DIS
LIN {X -44.405,Y 134.863,Z 176,A 109.661,B 6.9605,C 0.1314,E1 6.9122,E2 342.6563} C_DIS
LIN {X -47.7251,Y 133.7241,Z 176,A 111.0865,B 6.9605,C 0.1326,E1 6.9084,E2 341.2306} C_DIS
LIN {X -50.9888,Y 132.5141,Z 176,A 112.4991,B 6.9605,C 0.134,E1 6.9047,E2 339.8179} C_DIS
LIN {X -54.3435,Y 131.1737,Z 176,A 114.0023,B 6.9605,C 0.1349,E1 6.9008,E2 338.31} C_DIS
LIN {X -58.2643,Y 129.4796,Z 176,A 115.7197,B 6.9604,C 0.1369,E1 6.8964,E2 336.5947} C_DIS
LIN {X -61.342,Y 128.0498,Z 176,A 117.1086,B 6.9604,C 0.1383,E1 6.8929,E2 335.2043} C_DIS
LIN {X -64.5565,Y 126.4597,Z 176,A 118.5644,B 6.9604,C 0.1401,E1 6.8893,E2 333.7485} C_DIS
LIN {X -67.6382,Y 124.8414,Z 176,A 120.0045,B 6.9603,C 0.1415,E1 6.8857,E2 332.305} C_DIS
LIN {X -71.4422,Y 122.704,Z 176,A 121.7699,B 6.9603,C 0.1439,E1 6.8815,E2 330.5405} C_DIS
LIN {X -75.1653,Y 120.4589,Z 176,A 123.5463,B 6.9602,C 0.1462,E1 6.8772,E2 328.7626} C_DIS
LIN {X -78.8177,Y 118.1013,Z 176,A 125.2896,B 6.9602,C 0.1491,E1 6.8732,E2 327.0222} C_DIS
LIN {X -81.7363,Y 116.1006,Z 176,A 126.7407,B 6.9601,C 0.1512,E1 6.8698,E2 325.5694} C_DIS
LIN {X -84.6676,Y 113.9806,Z 176,A 128.3413,B 6.9601,C 0.1517,E1 6.8662,E2 323.9519} C_DIS
LIN {X -88.0027,Y 111.4262,Z 176,A 129.9532,B 6.96,C 0.1558,E1 6.8627,E2 322.3522} C_DIS
LIN {X -90.8913,Y 109.083,Z 176,A 131.593,B 6.96,C 0.1567,E1 6.8591,E2 320.6957} C_DIS
LIN {X -94.0261,Y 106.3919,Z 176,A 133.1502,B 6.9599,C 0.1613,E1 6.8558,E2 319.1542} C_DIS
LIN {X -96.6041,Y 104.0569,Z 176,A 134.5858,B 6.9599,C 0.1636,E1 6.8529,E2 317.7157} C_DIS
LIN {X -99.1696,Y 101.6153,Z 176,A 136.1487,B 6.9598,C 0.1647,E1 6.8497,E2 316.1369} C_DIS
LIN {X -102.1807,Y 98.5866,Z 176,A 137.7892,B 6.9597,C 0.1693,E1 6.8465,E2 314.5087} C_DIS
LIN {X -104.6638,Y 95.9461,Z 176,A 139.2638,B 6.9597,C 0.1723,E1 6.8437,E2 313.0338} C_DIS
LIN {X -106.9792,Y 93.3574,Z 176,A 140.682,B 6.9595,C 0.1751,E1 6.8411,E2 311.6147} C_DIS
LIN {X -109.2199,Y 90.726,Z 176,A 142.0934,B 6.9595,C 0.1779,E1 6.8386,E2 310.2025} C_DIS
LIN {X -111.3912,Y 88.0473,Z 176,A 143.5269,B 6.9594,C 0.1805,E1 6.8361,E2 308.7649} C_DIS
LIN {X -114.0045,Y 84.6355,Z 176,A 145.2946,B 6.9594,C 0.1841,E1 6.8331,E2 306.9945} C_DIS
LIN {X -116.1242,Y 81.7028,Z 176,A 146.9019,B 6.9593,C 0.1855,E1 6.8304,E2 305.3696} C_DIS
LIN {X -118.539,Y 78.1579,Z 176,A 148.516,B 6.9591,C 0.1912,E1 6.828,E2 303.7722} C_DIS
LIN {X -120.429,Y 75.2134,Z 176,A 149.9436,B 6.9591,C 0.1945,E1 6.8258,E2 302.3439} C_DIS
LIN {X -122.198,Y 72.3049,Z 176,A 151.4568,B 6.959,C 0.196,E1 6.8236,E2 300.8139} C_DIS
LIN {X -124.3586,Y 68.5213,Z 176,A 153.1687,B 6.9588,C 0.2011,E1 6.8213,E2 299.1097} C_DIS
LIN {X -126.0001,Y 65.4518,Z 176,A 154.5985,B 6.9588,C 0.2043,E1 6.8194,E2 297.6779} C_DIS
LIN {X -127.596,Y 62.283,Z 176,A 156.0615,B 6.9586,C 0.2076,E1 6.8176,E2 296.2122} C_DIS
LIN {X -129.1183,Y 59.0627,Z 176,A 157.5205,B 6.9586,C 0.2111,E1 6.8159,E2 294.7518} C_DIS
LIN {X -130.4785,Y 55.992,Z 176,A 158.8838,B 6.9584,C 0.2146,E1 6.8144,E2 293.3887} C_DIS
LIN {X -131.7625,Y 52.8987,Z 176,A 160.3001,B 6.9584,C 0.2173,E1 6.8129,E2 291.9653} C_DIS
LIN {X -133.0906,Y 49.4634,Z 176,A 161.7902,B 6.9582,C 0.2213,E1 6.8114,E2 290.4761} C_DIS
LIN {X -134.2628,Y 46.1868,Z 176,A 163.2221,B 6.9582,C 0.2248,E1 6.8101,E2 289.042} C_DIS
LIN {X -135.3544,Y 42.8826,Z 176,A 164.6381,B 6.958,C 0.2285,E1 6.8089,E2 287.6257} C_DIS
LIN {X -136.3264,Y 39.6835,Z 176,A 166.048,B 6.9579,C 0.2314,E1 6.8077,E2 286.2092} C_DIS
LIN {X -137.2934,Y 36.1983,Z 176,A 167.5195,B 6.9578,C 0.2353,E1 6.8067,E2 284.7374} C_DIS
LIN {X -138.0421,Y 33.2269,Z 176,A 168.8252,B 6.9577,C 0.2379,E1 6.8058,E2 283.4239} C_DIS
LIN {X -138.9069,Y 29.4086,Z 176,A 170.393,B 6.9575,C 0.2425,E1 6.8049,E2 281.8591} C_DIS
LIN {X -139.5954,Y 25.9482,Z 176,A 171.8409,B 6.9574,C 0.2462,E1 6.8041,E2 280.4094} C_DIS
LIN {X -140.1657,Y 22.6661,Z 176,A 173.2116,B 6.9573,C 0.2497,E1 6.8035,E2 279.0365} C_DIS
LIN {X -140.6779,Y 19.2366,Z 176,A 174.625,B 6.9571,C 0.2535,E1 6.8029,E2 277.6224} C_DIS
LIN {X -141.0459,Y 16.3097,Z 176,A 175.9742,B 6.9571,C 0.2549,E1 6.8025,E2 276.2535} C_DIS
LIN {X -141.4645,Y 12.1466,Z 176,A 177.5961,B 6.9569,C 0.2605,E1 6.802,E2 274.6418} C_DIS
LIN {X -141.7192,Y 8.6825,Z 176,A 179.0208,B 6.9567,C 0.2643,E1 6.8018,E2 273.2153} C_DIS
LIN {X -141.8841,Y 5.3544,Z 176,A -179.6431,B 6.9566,C 0.2682,E1 6.8016,E2 271.8815} C_DIS
LIN {X -141.9756,Y 1.7477,Z 176,A -178.1792,B 6.9564,C 0.2723,E1 6.8016,E2 270.4179} C_DIS
LIN {X -141.9781,Y -1.5992,Z 176,A -176.7018,B 6.9564,C 0.2746,E1 6.8016,E2 268.925} C_DIS
LIN {X -141.8881,Y -5.2504,Z 176,A -175.2229,B 6.9562,C 0.2787,E1 6.8016,E2 267.4465} C_DIS
LIN {X -141.7256,Y -8.5788,Z 176,A -173.9499,B 6.956,C 0.2835,E1 6.8019,E2 266.184} C_DIS
LIN {X -141.4753,Y -12.0187,Z 176,A -172.4166,B 6.9559,C 0.2857,E1 6.8022,E2 264.6333} C_DIS
LIN {X -141.1072,Y -15.7739,Z 176,A -170.8906,B 6.9557,C 0.29,E1 6.8027,E2 263.1081} C_DIS
LIN {X -140.6756,Y -19.2539,Z 176,A -169.4266,B 6.9556,C 0.2933,E1 6.8032,E2 261.6387} C_DIS
LIN {X -140.1691,Y -22.6459,Z 176,A -168.0439,B 6.9554,C 0.2973,E1 6.8038,E2 260.2572} C_DIS
LIN {X -139.6255,Y -25.7876,Z 176,A -166.6893,B 6.9553,C 0.3,E1 6.8045,E2 258.8947} C_DIS
LIN {X -138.9366,Y -29.2709,Z 176,A -165.2365,B 6.9551,C 0.3038,E1 6.8053,E2 257.4403} C_DIS
LIN {X -138.1446,Y -32.8015,Z 176,A -163.7494,B 6.955,C 0.3075,E1 6.8062,E2 255.9506} C_DIS
LIN {X -137.3785,Y -35.8792,Z 176,A -162.3875,B 6.9549,C 0.31,E1 6.8072,E2 254.5789} C_DIS
LIN {X -136.4046,Y -39.4165,Z 176,A -160.8984,B 6.9547,C 0.3139,E1 6.8083,E2 253.0897} C_DIS
LIN {X -135.3556,Y -42.879,Z 176,A -159.4841,B 6.9545,C 0.3185,E1 6.8095,E2 251.6823} C_DIS
LIN {X -134.3087,Y -46.0544,Z 176,A -158.0706,B 6.9543,C 0.3213,E1 6.8107,E2 250.2612} C_DIS
LIN {X -133.1351,Y -49.3445,Z 176,A -156.7718,B 6.9541,C 0.3265,E1 6.8119,E2 248.978} C_DIS
LIN {X -131.8871,Y -52.5895,Z 176,A -155.1676,B 6.9541,C 0.3275,E1 6.8136,E2 247.348} C_DIS
LIN {X -130.307,Y -56.3885,Z 176,A -153.4604,B 6.9539,C 0.3313,E1 6.8155,E2 245.6356} C_DIS
LIN {X -128.7218,Y -59.9199,Z 176,A -151.9222,B 6.9537,C 0.3356,E1 6.8173,E2 244.1015} C_DIS
LIN {X -127.2443,Y -62.9961,Z 176,A -150.5121,B 6.9535,C 0.3387,E1 6.819,E2 242.6877} C_DIS
LIN {X -125.6386,Y -66.1402,Z 176,A -149.1401,B 6.9533,C 0.3429,E1 6.8207,E2 241.3234} C_DIS
LIN {X -123.9233,Y -69.3056,Z 176,A -147.4541,B 6.9533,C 0.3434,E1 6.8231,E2 239.6074} C_DIS
LIN {X -121.7472,Y -73.0612,Z 176,A -145.6763,B 6.9531,C 0.3473,E1 6.8256,E2 237.827} C_DIS
LIN {X -119.4493,Y -76.7599,Z 176,A -143.8745,B 6.9529,C 0.3509,E1 6.8283,E2 236.0199} C_DIS
LIN {X -117.0799,Y -80.3272,Z 176,A -142.2694,B 6.9526,C 0.3566,E1 6.8308,E2 234.4319} C_DIS
LIN {X -115.1155,Y -83.1182,Z 176,A -140.8584,B 6.9525,C 0.3593,E1 6.8331,E2 233.017} C_DIS
LIN {X -113.0013,Y -85.9708,Z 176,A -139.4119,B 6.9523,C 0.3623,E1 6.8355,E2 231.5693} C_DIS
LIN {X -110.902,Y -88.6622,Z 176,A -137.9918,B 6.9523,C 0.3647,E1 6.838,E2 230.1441} C_DIS
LIN {X -108.7683,Y -91.2666,Z 176,A -136.5921,B 6.9521,C 0.3671,E1 6.8405,E2 228.7394} C_DIS
LIN {X -106.4081,Y -94.0078,Z 176,A -135.1362,B 6.9519,C 0.3702,E1 6.8431,E2 227.2844} C_DIS
LIN {X -104.0721,Y -96.5878,Z 176,A -133.6817,B 6.9519,C 0.3723,E1 6.8459,E2 225.8237} C_DIS
LIN {X -101.0643,Y -99.7313,Z 176,A -131.9024,B 6.9516,C 0.3755,E1 6.8494,E2 224.0417} C_DIS
LIN {X -97.9612,Y -102.7802,Z 176,A -130.1329,B 6.9515,C 0.3787,E1 6.8529,E2 222.2708} C_DIS
LIN {X -94.9272,Y -105.589,Z 176,A -128.3935,B 6.9514,C 0.3808,E1 6.8565,E2 220.5223} C_DIS
LIN {X -92.0771,Y -108.0831,Z 176,A -126.8942,B 6.9512,C 0.3839,E1 6.8597,E2 219.0272} C_DIS
LIN {X -88.7749,Y -110.8123,Z 176,A -125.1423,B 6.951,C 0.3866,E1 6.8635,E2 217.2725} C_DIS
LIN {X -85.975,Y -112.9981,Z 176,A -123.5611,B 6.951,C 0.3869,E1 6.867,E2 215.6716} C_DIS
LIN {X -82.4597,Y -115.5879,Z 176,A -121.9197,B 6.9508,C 0.3914,E1 6.8707,E2 214.0466} C_DIS
LIN {X -79.1005,Y -117.9125,Z 176,A -120.2,B 6.9507,C 0.3929,E1 6.8747,E2 212.3176} C_DIS
LIN {X -75.91,Y -119.991,Z 176,A -118.5762,B 6.9507,C 0.3939,E1 6.8785,E2 210.6822} C_DIS
LIN {X -72.3055,Y -122.1977,Z 176,A -116.9096,B 6.9505,C 0.3968,E1 6.8825,E2 209.0209} C_DIS
LIN {X -68.5046,Y -124.3679,Z 176,A -115.1834,B 6.9503,C 0.3997,E1 6.8867,E2 207.3} C_DIS
LIN {X -65.4359,Y -126.0085,Z 176,A -113.768,B 6.9503,C 0.4013,E1 6.8902,E2 205.8831} C_DIS
LIN {X -62.2103,Y -127.6319,Z 176,A -112.1585,B 6.9503,C 0.4007,E1 6.8943,E2 204.253} C_DIS
LIN {X -58.1955,Y -129.5103,Z 176,A -110.4032,B 6.9501,C 0.4031,E1 6.8987,E2 202.502} C_DIS
LIN {X -54.4646,Y -131.1231,Z 176,A -108.8515,B 6.9499,C 0.4061,E1 6.9027,E2 200.9621} C_DIS
LIN {X -51.3388,Y -132.378,Z 176,A -107.4955,B 6.9499,C 0.4075,E1 6.9062,E2 199.6063} C_DIS
LIN {X -47.8352,Y -133.6844,Z 176,A -105.9656,B 6.9498,C 0.4085,E1 6.9102,E2 198.0733} C_DIS
LIN {X -44.5447,Y -134.8165,Z 176,A -104.5533,B 6.9498,C 0.4095,E1 6.914,E2 196.6597} C_DIS
LIN {X -41.356,Y -135.8284,Z 176,A -103.2677,B 6.9496,C 0.4114,E1 6.9174,E2 195.3826} C_DIS
LIN {X -37.8544,Y -136.846,Z 176,A -101.7199,B 6.9496,C 0.4113,E1 6.9216,E2 193.8242} C_DIS
LIN {X -34.4988,Y -137.7304,Z 176,A -100.3269,B 6.9496,C 0.4122,E1 6.9253,E2 192.4318} C_DIS
LIN {X -31.2358,Y -138.5068,Z 176,A -98.9642,B 6.9496,C 0.4128,E1 6.9291,E2 191.0675} C_DIS
LIN {X -27.6994,Y -139.258,Z 176,A -97.496,B 6.9496,C 0.4133,E1 6.9331,E2 189.5976} C_DIS
LIN {X -24.2795,Y -139.8954,Z 176,A -96.0941,B 6.9495,C 0.4139,E1 6.9369,E2 188.1955} C_DIS
LIN {X -20.9644,Y -140.4307,Z 176,A -94.7269,B 6.9495,C 0.4141,E1 6.9407,E2 186.8263} C_DIS
LIN {X -17.5454,Y -140.8985,Z 176,A -93.3035,B 6.9495,C 0.414,E1 6.9447,E2 185.3982} C_DIS
LIN {X -14.0553,Y -141.2883,Z 176,A -91.8661,B 6.9495,C 0.414,E1 6.9487,E2 183.9575} C_DIS
LIN {X -10.4522,Y -141.5997,Z 176,A -90.4428,B 6.9495,C 0.4147,E1 6.9526,E2 182.5385} C_DIS
LIN {X -6.9596,Y -141.8144,Z 176,A -89.0597,B 6.9494,C 0.4152,E1 6.9565,E2 181.1587} C_DIS
LIN {X -3.6178,Y -141.9393,Z 176,A -87.6878,B 6.9494,C 0.4148,E1 6.9603,E2 179.7832} C_DIS
LIN {X -0.1384,Y -141.9864,Z 176,A -86.2539,B 6.9494,C 0.4141,E1 6.9643,E2 178.3447} C_DIS
LIN {X -0.1384,Y -141.9864,Z 176,A -86.2539,B 6.9494,C 0.4141,E1 6.9643,E2 178.3447} C_DIS
Enddeposition()
LIN {X 0.9633,Y -133.0465,Z 177,A -86.3117,B 6.5192,C 0.3825,E1 6.5331,E2 178.2616} C_DIS
Startdeposition()
$VEL.CP = VEL_PRINT
LIN {X -1.7457,Y -133.0408,Z 177,A -87.6946,B 6.519,C 0.3857,E1 6.5292,E2 179.6721} C_DIS
LIN {X -5.0028,Y -132.9575,Z 177,A -89.0941,B 6.519,C 0.3857,E1 6.5253,E2 181.0717} C_DIS
LIN {X -8.2598,Y -132.7948,Z 177,A -90.512,B 6.519,C 0.3858,E1 6.5213,E2 182.4918} C_DIS
LIN {X -11.5127,Y -132.5527,Z 177,A -91.9125,B 6.519,C 0.3856,E1 6.5174,E2 183.8924} C_DIS
LIN {X -14.7748,Y -132.2295,Z 177,A -93.322,B 6.519,C 0.3853,E1 6.5135,E2 185.3022} C_DIS
LIN {X -18.0134,Y -131.8283,Z 177,A -94.7272,B 6.519,C 0.385,E1 6.5096,E2 186.7079} C_DIS
LIN {X -21.1424,Y -131.3629,Z 177,A -96.121,B 6.519,C 0.385,E1 6.5057,E2 188.1061} C_DIS
LIN {X -24.356,Y -130.8045,Z 177,A -97.5257,B 6.5191,C 0.3845,E1 6.5019,E2 189.5113} C_DIS
LIN {X -27.5567,Y -130.1673,Z 177,A -99.0508,B 6.5191,C 0.3854,E1 6.4977,E2 191.0516} C_DIS
LIN {X -31.9494,Y -129.1606,Z 177,A -101.027,B 6.5191,C 0.3848,E1 6.4923,E2 193.0327} C_DIS
LIN {X -35.6573,Y -128.1842,Z 177,A -102.5061,B 6.5193,C 0.3815,E1 6.4883,E2 194.4908} C_DIS
LIN {X -38.7504,Y -127.2832,Z 177,A -103.9046,B 6.5193,C 0.3807,E1 6.4846,E2 195.891} C_DIS
LIN {X -42.3117,Y -126.1443,Z 177,A -105.5992,B 6.5193,C 0.3805,E1 6.4801,E2 197.5963} C_DIS
LIN {X -46.3658,Y -124.7112,Z 177,A -107.4404,B 6.5195,C 0.3788,E1 6.4752,E2 199.4366} C_DIS
LIN {X -49.4989,Y -123.501,Z 177,A -108.8724,B 6.5195,C 0.3773,E1 6.4715,E2 200.867} C_DIS
LIN {X -52.424,Y -122.2883,Z 177,A -110.3607,B 6.5195,C 0.3775,E1 6.4676,E2 202.3709} C_DIS
LIN {X -55.4087,Y -120.9655,Z 177,A -111.7482,B 6.5196,C 0.3757,E1 6.4641,E2 203.7563} C_DIS
LIN {X -58.3588,Y -119.5705,Z 177,A -113.0766,B 6.5198,C 0.3732,E1 6.4608,E2 205.0753} C_DIS
LIN {X -61.2733,Y -118.1039,Z 177,A -114.6051,B 6.5198,C 0.373,E1 6.457,E2 206.6191} C_DIS
LIN {X -64.6367,Y -116.298,Z 177,A -116.0398,B 6.52,C 0.3683,E1 6.4535,E2 208.0281} C_DIS
LIN {X -67.0903,Y -114.9004,Z 177,A -117.3852,B 6.52,C 0.3683,E1 6.4502,E2 209.3894} C_DIS
LIN {X -69.802,Y -113.2733,Z 177,A -118.7716,B 6.5201,C 0.3667,E1 6.4469,E2 210.7788} C_DIS
LIN {X -72.6392,Y -111.475,Z 177,A -120.2344,B 6.5202,C 0.3648,E1 6.4435,E2 212.2435} C_DIS
LIN {X -75.3766,Y -109.6424,Z 177,A -121.6668,B 6.5204,C 0.3629,E1 6.4401,E2 213.6775} C_DIS
LIN {X -78.032,Y -107.7687,Z 177,A -123.1495,B 6.5204,C 0.3617,E1 6.4367,E2 215.1703} C_DIS
LIN {X -81.2127,Y -105.3931,Z 177,A -124.8834,B 6.5206,C 0.3592,E1 6.4329,E2 216.907} C_DIS
LIN {X -84.4485,Y -102.8184,Z 177,A -126.7772,B 6.5206,C 0.3574,E1 6.4287,E2 218.8144} C_DIS
LIN {X -87.5241,Y -100.2128,Z 177,A -128.3935,B 6.5209,C 0.3529,E1 6.4253,E2 220.4157} C_DIS
LIN {X -90.5275,Y -97.5084,Z 177,A -130.1663,B 6.5211,C 0.3501,E1 6.4217,E2 222.1921} C_DIS
LIN {X -93.5068,Y -94.6557,Z 177,A -131.9555,B 6.5212,C 0.3468,E1 6.4181,E2 223.9825} C_DIS
LIN {X -96.3625,Y -91.7464,Z 177,A -133.7458,B 6.5214,C 0.3438,E1 6.4146,E2 225.7766} C_DIS
LIN {X -99.1478,Y -88.7287,Z 177,A -135.6865,B 6.5214,C 0.3421,E1 6.4109,E2 227.7378} C_DIS
LIN {X -101.8389,Y -85.6267,Z 177,A -137.4668,B 6.5217,C 0.3385,E1 6.4077,E2 229.519} C_DIS
LIN {X -104.3976,Y -82.4885,Z 177,A -139.1104,B 6.5219,C 0.3336,E1 6.4048,E2 231.1498} C_DIS
LIN {X -106.8722,Y -79.2557,Z 177,A -140.8921,B 6.5221,C 0.33,E1 6.4018,E2 232.9344} C_DIS
LIN {X -108.7809,Y -76.6146,Z 177,A -142.3832,B 6.5222,C 0.3278,E1 6.3994,E2 234.4356} C_DIS
LIN {X -110.6314,Y -73.9174,Z 177,A -143.894,B 6.5223,C 0.3257,E1 6.397,E2 235.9582} C_DIS
LIN {X -112.4625,Y -71.1005,Z 177,A -145.1996,B 6.5226,C 0.3207,E1 6.3951,E2 237.2461} C_DIS
LIN {X -114.1507,Y -68.3577,Z 177,A -146.6582,B 6.5226,C 0.3182,E1 6.393,E2 238.7128} C_DIS
LIN {X -115.8313,Y -65.4698,Z 177,A -148.0996,B 6.5228,C 0.3147,E1 6.3909,E2 240.1538} C_DIS
LIN {X -117.395,Y -62.623,Z 177,A -149.5514,B 6.523,C 0.3118,E1 6.389,E2 241.6114} C_DIS
LIN {X -118.9692,Y -59.5776,Z 177,A -151.1199,B 6.5231,C 0.3091,E1 6.387,E2 243.1903} C_DIS
LIN {X -120.3205,Y -56.797,Z 177,A -152.4031,B 6.5233,C 0.3052,E1 6.3855,E2 244.4669} C_DIS
LIN {X -121.7758,Y -53.6079,Z 177,A -153.9393,B 6.5235,C 0.3016,E1 6.3837,E2 246.0055} C_DIS
LIN {X -122.9236,Y -50.9164,Z 177,A -155.228,B 6.5235,C 0.2986,E1 6.3823,E2 247.2969} C_DIS
LIN {X -124.1743,Y -47.7859,Z 177,A -156.7086,B 6.5238,C 0.2951,E1 6.3808,E2 248.7802} C_DIS
LIN {X -125.275,Y -44.8201,Z 177,A -158.099,B 6.5239,C 0.2918,E1 6.3795,E2 250.1732} C_DIS
LIN {X -126.3667,Y -41.6437,Z 177,A -159.6441,B 6.524,C 0.289,E1 6.3781,E2 251.7293} C_DIS
LIN {X -127.3495,Y -38.534,Z 177,A -161.1357,B 6.5242,C 0.2861,E1 6.3769,E2 253.2305} C_DIS
LIN {X -128.3006,Y -35.2408,Z 177,A -162.5152,B 6.5244,C 0.281,E1 6.3758,E2 254.5975} C_DIS
LIN {X -129.1055,Y -32.1668,Z 177,A -163.9058,B 6.5245,C 0.2775,E1 6.3749,E2 255.9898} C_DIS
LIN {X -129.9517,Y -28.5551,Z 177,A -165.4231,B 6.5247,C 0.2722,E1 6.3739,E2 257.4964} C_DIS
LIN {X -130.5157,Y -25.8597,Z 177,A -166.7549,B 6.5248,C 0.2704,E1 6.3732,E2 258.8449} C_DIS
LIN {X -131.111,Y -22.652,Z 177,A -168.2145,B 6.525,C 0.2671,E1 6.3724,E2 260.3101} C_DIS
LIN {X -131.6128,Y -19.5249,Z 177,A -169.6094,B 6.5251,C 0.2636,E1 6.3718,E2 261.7078} C_DIS
LIN {X -132.0523,Y -16.2826,Z 177,A -171.0483,B 6.5252,C 0.2599,E1 6.3713,E2 263.1492} C_DIS
LIN {X -132.4112,Y -13.0397,Z 177,A -172.481,B 6.5254,C 0.2562,E1 6.3709,E2 264.5841} C_DIS
LIN {X -132.6909,Y -9.7879,Z 177,A -173.9305,B 6.5255,C 0.2526,E1 6.3706,E2 266.0378} C_DIS
LIN {X -132.8912,Y -6.5299,Z 177,A -175.3546,B 6.5257,C 0.2488,E1 6.3704,E2 267.4631} C_DIS
LIN {X -133.0122,Y -3.2594,Z 177,A -176.8449,B 6.5257,C 0.2457,E1 6.3702,E2 268.9619} C_DIS
LIN {X -133.0519,Y 0.5181,Z 177,A -178.399,B 6.526,C 0.2402,E1 6.3702,E2 270.5061} C_DIS
LIN {X -133.0121,Y 3.2656,Z 177,A -179.704,B 6.526,C 0.2381,E1 6.3702,E2 271.8246} C_DIS
LIN {X -132.8913,Y 6.5268,Z 177,A 178.8734,B 6.5262,C 0.2343,E1 6.3705,E2 273.2481} C_DIS
LIN {X -132.6242,Y 10.666,Z 177,A 176.8913,B 6.5263,C 0.2312,E1 6.3709,E2 275.2521} C_DIS
LIN {X -132.2309,Y 14.7625,Z 177,A 175.2681,B 6.5266,C 0.2246,E1 6.3713,E2 276.8561} C_DIS
LIN {X -131.8299,Y 18.001,Z 177,A 173.7782,B 6.5266,C 0.2215,E1 6.3719,E2 278.3549} C_DIS
LIN {X -131.3643,Y 21.1338,Z 177,A 172.4099,B 6.5268,C 0.2177,E1 6.3724,E2 279.7225} C_DIS
LIN {X -130.8054,Y 24.3511,Z 177,A 170.9763,B 6.5269,C 0.214,E1 6.3732,E2 281.1581} C_DIS
LIN {X -130.1635,Y 27.5742,Z 177,A 169.5037,B 6.527,C 0.2106,E1 6.374,E2 282.6363} C_DIS
LIN {X -129.4488,Y 30.7537,Z 177,A 168.0984,B 6.5271,C 0.2067,E1 6.3749,E2 284.0406} C_DIS
LIN {X -128.6311,Y 34.0103,Z 177,A 166.622,B 6.5273,C 0.203,E1 6.3759,E2 285.5193} C_DIS
LIN {X -127.7859,Y 37.0601,Z 177,A 165.2039,B 6.5273,C 0.1998,E1 6.377,E2 286.9427} C_DIS
LIN {X -126.8389,Y 40.1818,Z 177,A 163.7694,B 6.5275,C 0.1963,E1 6.3782,E2 288.3796} C_DIS
LIN {X -125.7841,Y 43.3702,Z 177,A 162.3426,B 6.5275,C 0.1922,E1 6.3794,E2 289.8027} C_DIS
LIN {X -124.7046,Y 46.3832,Z 177,A 160.891,B 6.5277,C 0.1892,E1 6.3808,E2 291.2618} C_DIS
LIN {X -123.3984,Y 49.7533,Z 177,A 159.257,B 6.5277,C 0.1859,E1 6.3825,E2 292.9035} C_DIS
LIN {X -122.1312,Y 52.7874,Z 177,A 157.9355,B 6.5279,C 0.1811,E1 6.384,E2 294.2125} C_DIS
LIN {X -120.9372,Y 55.4698,Z 177,A 156.5979,B 6.5279,C 0.1786,E1 6.3855,E2 295.5577} C_DIS
LIN {X -119.5662,Y 58.3674,Z 177,A 155.1788,B 6.5281,C 0.1754,E1 6.3872,E2 296.9802} C_DIS
LIN {X -118.1002,Y 61.2805,Z 177,A 153.7642,B 6.5281,C 0.172,E1 6.389,E2 298.3947} C_DIS
LIN {X -116.5639,Y 64.1565,Z 177,A 152.3122,B 6.5282,C 0.1689,E1 6.3909,E2 299.8511} C_DIS
LIN {X -114.9091,Y 67.0754,Z 177,A 150.8374,B 6.5283,C 0.1657,E1 6.393,E2 301.3281} C_DIS
LIN {X -113.2815,Y 69.7886,Z 177,A 149.44,B 6.5283,C 0.1627,E1 6.395,E2 302.7284} C_DIS
LIN {X -111.4852,Y 72.6234,Z 177,A 147.9677,B 6.5285,C 0.1595,E1 6.3973,E2 304.2026} C_DIS
LIN {X -109.6595,Y 75.3517,Z 177,A 146.527,B 6.5285,C 0.1564,E1 6.3995,E2 305.6451} C_DIS
LIN {X -107.7742,Y 78.0244,Z 177,A 145.0965,B 6.5286,C 0.1534,E1 6.4018,E2 307.0769} C_DIS
LIN {X -105.3912,Y 81.2151,Z 177,A 143.3416,B 6.5286,C 0.1499,E1 6.4048,E2 308.835} C_DIS
LIN {X -102.8521,Y 84.4073,Z 177,A 141.404,B 6.5287,C 0.148,E1 6.4082,E2 310.7923} C_DIS
LIN {X -100.2102,Y 87.5271,Z 177,A 139.7247,B 6.5288,C 0.1432,E1 6.4113,E2 312.4605} C_DIS
LIN {X -97.48,Y 90.5579,Z 177,A 137.9747,B 6.5289,C 0.1394,E1 6.4146,E2 314.2082} C_DIS
LIN {X -94.6589,Y 93.5036,Z 177,A 136.1912,B 6.5289,C 0.1361,E1 6.418,E2 315.9933} C_DIS
LIN {X -91.748,Y 96.361,Z 177,A 134.3993,B 6.5291,C 0.133,E1 6.4216,E2 317.7878} C_DIS
LIN {X -88.7441,Y 99.134,Z 177,A 132.4762,B 6.5291,C 0.1315,E1 6.4256,E2 319.7285} C_DIS
LIN {X -85.6267,Y 101.8389,Z 177,A 130.6894,B 6.5291,C 0.1283,E1 6.4294,E2 321.5148} C_DIS
LIN {X -82.503,Y 104.3862,Z 177,A 129.0523,B 6.5292,C 0.1241,E1 6.433,E2 323.1389} C_DIS
LIN {X -79.257,Y 106.8712,Z 177,A 127.2627,B 6.5292,C 0.1214,E1 6.437,E2 324.9305} C_DIS
LIN {X -76.5744,Y 108.8093,Z 177,A 125.8315,B 6.5293,C 0.1191,E1 6.4402,E2 326.3612} C_DIS
LIN {X -73.3198,Y 111.0285,Z 177,A 124.2243,B 6.5293,C 0.1153,E1 6.4439,E2 327.9566} C_DIS
LIN {X -71.0872,Y 112.4708,Z 177,A 122.9822,B 6.5293,C 0.1147,E1 6.4469,E2 329.2092} C_DIS
LIN {X -68.2885,Y 114.1919,Z 177,A 121.4778,B 6.5294,C 0.1137,E1 6.4505,E2 330.723} C_DIS
LIN {X -65.5024,Y 115.8129,Z 177,A 119.9746,B 6.5294,C 0.1131,E1 6.4541,E2 332.2386} C_DIS
LIN {X -62.6272,Y 117.3928,Z 177,A 118.6769,B 6.5294,C 0.1098,E1 6.4573,E2 333.5217} C_DIS
LIN {X -59.4408,Y 119.0367,Z 177,A 117.1982,B 6.5295,C 0.107,E1 6.461,E2 334.9916} C_DIS
LIN {X -56.798,Y 120.32,Z 177,A 115.8492,B 6.5295,C 0.1065,E1 6.4644,E2 336.3495} C_DIS
LIN {X -53.8227,Y 121.6797,Z 177,A 114.4361,B 6.5295,C 0.1049,E1 6.468,E2 337.7621} C_DIS
LIN {X -50.8966,Y 122.9319,Z 177,A 113.0479,B 6.5295,C 0.1036,E1 6.4716,E2 339.1513} C_DIS
LIN {X -47.7747,Y 124.1787,Z 177,A 111.5898,B 6.5296,C 0.1022,E1 6.4753,E2 340.6096} C_DIS
LIN {X -44.6873,Y 125.3229,Z 177,A 110.1744,B 6.5296,C 0.1008,E1 6.4791,E2 342.0237} C_DIS
LIN {X -41.6448,Y 126.3664,Z 177,A 108.7774,B 6.5296,C 0.0997,E1 6.4828,E2 343.4212} C_DIS
LIN {X -38.0719,Y 127.4897,Z 177,A 107.1828,B 6.5296,C 0.0982,E1 6.487,E2 345.0126} C_DIS
LIN {X -35.4825,Y 128.233,Z 177,A 105.9694,B 6.5296,C 0.0979,E1 6.4903,E2 346.2315} C_DIS
LIN {X -32.2341,Y 129.0884,Z 177,A 104.5334,B 6.5296,C 0.0968,E1 6.4942,E2 347.6654} C_DIS
LIN {X -29.0435,Y 129.8439,Z 177,A 103.1096,B 6.5296,C 0.0961,E1 6.498,E2 349.0897} C_DIS
LIN {X -25.8535,Y 130.517,Z 177,A 101.7022,B 6.5297,C 0.0953,E1 6.5019,E2 350.4967} C_DIS
LIN {X -22.644,Y 131.1124,Z 177,A 100.2703,B 6.5297,C 0.095,E1 6.5058,E2 351.9309} C_DIS
LIN {X -19.5212,Y 131.6133,Z 177,A 98.9016,B 6.5297,C 0.0945,E1 6.5096,E2 353.2996} C_DIS
LIN {X -16.0906,Y 132.0752,Z 177,A 97.4678,B 6.5297,C 0.0932,E1 6.5136,E2 354.7259} C_DIS
LIN {X -12.661,Y 132.4476,Z 177,A 96.0109,B 6.5297,C 0.0924,E1 6.5176,E2 356.1787} C_DIS
LIN {X -8.8655,Y 132.7575,Z 177,A 94.1154,B 6.5297,C 0.0955,E1 6.523,E2 358.1034} C_DIS
LIN {X -4.8,Y 132.9654,Z 177,A 92.3915,B 6.5297,C 0.0949,E1 6.5278,E2 359.8229} C_DIS
LIN {X -1.6189,Y 133.0429,Z 177,A 91.1499,B 6.5297,C 0.0932,E1 6.5312,E2 361.0488} C_DIS
LIN {X 1.7385,Y 133.041,Z 177,A 89.7309,B 6.5297,C 0.0929,E1 6.5351,E2 362.4641} C_DIS
LIN {X 5.4619,Y 132.9396,Z 177,A 88.2127,B 6.5297,C 0.0919,E1 6.5393,E2 363.9715} C_DIS
LIN {X 8.2562,Y 132.795,Z 177,A 86.9157,B 6.5297,C 0.0933,E1 6.543,E2 365.2789} C_DIS
LIN {X 11.5212,Y 132.552,Z 177,A 85.514,B 6.5297,C 0.0936,E1 6.5469,E2 366.6791} C_DIS
LIN {X 14.7688,Y 132.2302,Z 177,A 84.1159,B 6.5297,C 0.0939,E1 6.5508,E2 368.0758} C_DIS
LIN {X 18.4218,Y 131.7704,Z 177,A 82.6806,B 6.5297,C 0.0925,E1 6.5547,E2 369.493} C_DIS
LIN {X 21.1394,Y 131.3634,Z 177,A 81.3319,B 6.5297,C 0.0953,E1 6.5585,E2 370.8608} C_DIS
LIN {X 24.3545,Y 130.8048,Z 177,A 79.9362,B 6.5297,C 0.0959,E1 6.5623,E2 372.255} C_DIS
LIN {X 27.5579,Y 130.167,Z 177,A 78.5094,B 6.5297,C 0.097,E1 6.5662,E2 373.6836} C_DIS
LIN {X 30.8825,Y 129.4178,Z 177,A 77.0959,B 6.5297,C 0.0972,E1 6.57,E2 375.0904} C_DIS
LIN {X 34.0614,Y 128.6175,Z 177,A 75.6829,B 6.5297,C 0.0983,E1 6.5739,E2 376.5033} C_DIS
LIN {X 37.0816,Y 127.7797,Z 177,A 74.2263,B 6.5297,C 0.1009,E1 6.5778,E2 377.9722} C_DIS
LIN {X 41.3328,Y 126.4702,Z 177,A 72.2894,B 6.5296,C 0.1029,E1 6.583,E2 379.9112} C_DIS
LIN {X 44.8312,Y 125.271,Z 177,A 70.8564,B 6.5296,C 0.1021,E1 6.5867,E2 381.3252} C_DIS
LIN {X 47.9802,Y 124.0988,Z 177,A 69.4208,B 6.5296,C 0.1034,E1 6.5904,E2 382.7592} C_DIS
LIN {X 51.5951,Y 122.6402,Z 177,A 67.9056,B 6.5296,C 0.1028,E1 6.5943,E2 384.255} C_DIS
LIN {X 54.2154,Y 121.5041,Z 177,A 66.6299,B 6.5296,C 0.1049,E1 6.5976,E2 385.536} C_DIS
LIN {X 56.8846,Y 120.2786,Z 177,A 65.289,B 6.5296,C 0.1076,E1 6.601,E2 386.8858} C_DIS
LIN {X 59.8216,Y 118.8456,Z 177,A 63.8931,B 6.5295,C 0.1092,E1 6.6045,E2 388.2803} C_DIS
LIN {X 62.8727,Y 117.2609,Z 177,A 62.469,B 6.5295,C 0.1104,E1 6.608,E2 389.6977} C_DIS
LIN {X 65.5901,Y 115.7634,Z 177,A 61.0838,B 6.5295,C 0.113,E1 6.6114,E2 391.0888} C_DIS
LIN {X 68.4895,Y 114.0721,Z 177,A 59.5983,B 6.5294,C 0.1157,E1 6.615,E2 392.579} C_DIS
LIN {X 71.1847,Y 112.4093,Z 177,A 58.2909,B 6.5294,C 0.117,E1 6.6181,E2 393.8798} C_DIS
LIN {X 74.0735,Y 110.5271,Z 177,A 56.8627,B 6.5294,C 0.1185,E1 6.6214,E2 395.3014} C_DIS
LIN {X 76.7148,Y 108.7102,Z 177,A 55.3827,B 6.5293,C 0.1222,E1 6.6248,E2 396.7933} C_DIS
LIN {X 79.3431,Y 106.8072,Z 177,A 53.992,B 6.5293,C 0.1245,E1 6.6279,E2 398.1835} C_DIS
LIN {X 82.5421,Y 104.3553,Z 177,A 52.2547,B 6.5292,C 0.1276,E1 6.6317,E2 399.9212} C_DIS
LIN {X 86.2505,Y 101.3111,Z 177,A 50.3574,B 6.5292,C 0.1288,E1 6.6358,E2 401.7989} C_DIS
LIN {X 88.7918,Y 99.0913,Z 177,A 48.806,B 6.5291,C 0.1331,E1 6.639,E2 403.3621} C_DIS
LIN {X 91.7841,Y 96.3265,Z 177,A 47.0738,B 6.529,C 0.1362,E1 6.6425,E2 405.0921} C_DIS
LIN {X 94.6906,Y 93.4716,Z 177,A 45.3277,B 6.529,C 0.1396,E1 6.646,E2 406.8377} C_DIS
LIN {X 97.5166,Y 90.5186,Z 177,A 43.6028,B 6.5288,C 0.1427,E1 6.6493,E2 408.5589} C_DIS
LIN {X 100.7204,Y 86.9395,Z 177,A 41.6769,B 6.5288,C 0.1449,E1 6.6528,E2 410.4685} C_DIS
LIN {X 103.404,Y 83.7303,Z 177,A 39.8133,B 6.5287,C 0.1498,E1 6.6561,E2 412.34} C_DIS
LIN {X 106.2175,Y 80.1307,Z 177,A 38.0347,B 6.5287,C 0.1513,E1 6.6591,E2 414.0969} C_DIS
LIN {X 107.8391,Y 77.9347,Z 177,A 36.8556,B 6.5286,C 0.154,E1 6.6611,E2 415.2768} C_DIS
LIN {X 109.7162,Y 75.269,Z 177,A 35.4028,B 6.5285,C 0.1581,E1 6.6634,E2 416.7361} C_DIS
LIN {X 111.5812,Y 72.4756,Z 177,A 34.0264,B 6.5285,C 0.1604,E1 6.6655,E2 418.1047} C_DIS
LIN {X 113.2752,Y 69.7988,Z 177,A 32.7263,B 6.5284,C 0.1627,E1 6.6674,E2 419.3977} C_DIS
LIN {X 115.0007,Y 66.9179,Z 177,A 31.3076,B 6.5284,C 0.1658,E1 6.6694,E2 420.8138} C_DIS
LIN {X 116.8808,Y 63.5765,Z 177,A 29.5872,B 6.5282,C 0.1711,E1 6.6718,E2 422.5433} C_DIS
LIN {X 118.309,Y 60.8755,Z 177,A 28.4829,B 6.5282,C 0.1709,E1 6.6732,E2 423.623} C_DIS
LIN {X 119.615,Y 58.2685,Z 177,A 27.1557,B 6.5281,C 0.1753,E1 6.6748,E2 424.9594} C_DIS
LIN {X 121.008,Y 55.3167,Z 177,A 25.78,B 6.528,C 0.1785,E1 6.6764,E2 426.3322} C_DIS
LIN {X 122.3161,Y 52.3598,Z 177,A 24.4188,B 6.5279,C 0.1816,E1 6.6779,E2 427.6905} C_DIS
LIN {X 123.5507,Y 49.3755,Z 177,A 23.047,B 6.5278,C 0.1849,E1 6.6794,E2 429.0607} C_DIS
LIN {X 124.7538,Y 46.252,Z 177,A 21.6542,B 6.5278,C 0.188,E1 6.6808,E2 430.4486} C_DIS
LIN {X 126.0442,Y 42.6122,Z 177,A 20.0951,B 6.5276,C 0.1908,E1 6.6822,E2 431.9962} C_DIS
LIN {X 126.8958,Y 40.0036,Z 177,A 18.8675,B 6.5276,C 0.1947,E1 6.6832,E2 433.23} C_DIS
LIN {X 127.7868,Y 37.0571,Z 177,A 17.5636,B 6.5274,C 0.198,E1 6.6843,E2 434.5322} C_DIS
LIN {X 128.6823,Y 33.8183,Z 177,A 16.0689,B 6.5273,C 0.2028,E1 6.6854,E2 436.0336} C_DIS
LIN {X 129.4526,Y 30.7382,Z 177,A 14.6667,B 6.5271,C 0.2072,E1 6.6863,E2 437.441} C_DIS
LIN {X 130.1888,Y 27.4571,Z 177,A 13.3983,B 6.5271,C 0.2082,E1 6.687,E2 438.6887} C_DIS
LIN {X 130.9193,Y 23.7244,Z 177,A 11.9769,B 6.5271,C 0.2092,E1 6.6878,E2 440.085} C_DIS
LIN {X 131.3785,Y 21.0429,Z 177,A 10.6583,B 6.5269,C 0.215,E1 6.6884,E2 441.4224} C_DIS
LIN {X 131.8433,Y 17.8987,Z 177,A 9.2916,B 6.5267,C 0.2188,E1 6.6889,E2 442.7898} C_DIS
LIN {X 132.2417,Y 14.662,Z 177,A 7.9202,B 6.5267,C 0.2222,E1 6.6894,E2 444.1583} C_DIS
LIN {X 132.5609,Y 11.4153,Z 177,A 6.5505,B 6.5265,C 0.2256,E1 6.6897,E2 445.5248} C_DIS
LIN {X 132.8439,Y 7.4631,Z 177,A 4.6654,B 6.5262,C 0.2335,E1 6.69,E2 447.4329} C_DIS
LIN {X 133.0122,Y 3.2597,Z 177,A 3.0629,B 6.5262,C 0.2352,E1 6.6902,E2 449.0115} C_DIS
LIN {X 133.0518,Y -0.5293,Z 177,A 1.5755,B 6.5262,C 0.2374,E1 6.6902,E2 450.4827} C_DIS
LIN {X 133.0121,Y -3.264,Z 177,A 0.3307,B 6.5259,C 0.2419,E1 6.6902,E2 451.7366} C_DIS
LIN {X 132.8908,Y -6.5375,Z 177,A -1.0345,B 6.5259,C 0.2452,E1 6.69,E2 453.0975} C_DIS
LIN {X 132.6834,Y -9.8911,Z 177,A -2.423,B 6.5257,C 0.2484,E1 6.6897,E2 454.48} C_DIS
LIN {X 132.4015,Y -13.1412,Z 177,A -3.7926,B 6.5256,C 0.2518,E1 6.6894,E2 455.8465} C_DIS
LIN {X 132.0402,Y -16.3841,Z 177,A -5.1647,B 6.5254,C 0.2552,E1 6.6889,E2 457.2158} C_DIS
LIN {X 131.6134,Y -19.5207,Z 177,A -6.5001,B 6.5253,C 0.2586,E1 6.6884,E2 458.5491} C_DIS
LIN {X 131.0934,Y -22.7513,Z 177,A -7.8998,B 6.5251,C 0.2625,E1 6.6877,E2 459.9489} C_DIS
LIN {X 130.4955,Y -25.9593,Z 177,A -9.2841,B 6.525,C 0.2661,E1 6.687,E2 461.3319} C_DIS
LIN {X 129.8186,Y -29.1545,Z 177,A -10.7104,B 6.5248,C 0.2704,E1 6.6862,E2 462.7617} C_DIS
LIN {X 129.0341,Y -32.4482,Z 177,A -12.082,B 6.5248,C 0.273,E1 6.6853,E2 464.1241} C_DIS
LIN {X 128.1938,Y -35.623,Z 177,A -13.4237,B 6.5246,C 0.2757,E1 6.6843,E2 465.4582} C_DIS
LIN {X 127.2915,Y -38.7233,Z 177,A -14.8368,B 6.5244,C 0.28,E1 6.6832,E2 466.8754} C_DIS
LIN {X 126.303,Y -41.8351,Z 177,A -16.1893,B 6.5243,C 0.2829,E1 6.682,E2 468.2226} C_DIS
LIN {X 125.2729,Y -44.8259,Z 177,A -17.5221,B 6.5242,C 0.2861,E1 6.6808,E2 469.553} C_DIS
LIN {X 124.0989,Y -47.9799,Z 177,A -18.9411,B 6.524,C 0.2896,E1 6.6794,E2 470.9696} C_DIS
LIN {X 122.8853,Y -51.0083,Z 177,A -20.2899,B 6.5239,C 0.2924,E1 6.6779,E2 472.3129} C_DIS
LIN {X 121.637,Y -53.9183,Z 177,A -21.6503,B 6.5237,C 0.296,E1 6.6764,E2 473.6742} C_DIS
LIN {X 120.2786,Y -56.8847,Z 177,A -23.0254,B 6.5236,C 0.2992,E1 6.6748,E2 475.047} C_DIS
LIN {X 118.8483,Y -59.8163,Z 177,A -24.3999,B 6.5234,C 0.3023,E1 6.6731,E2 476.419} C_DIS
LIN {X 117.3482,Y -62.7101,Z 177,A -25.9137,B 6.5232,C 0.3078,E1 6.6711,E2 477.9478} C_DIS
LIN {X 115.7643,Y -65.5885,Z 177,A -27.1914,B 6.5232,C 0.3091,E1 6.6694,E2 479.2099} C_DIS
LIN {X 114.0714,Y -68.4906,Z 177,A -28.5838,B 6.523,C 0.3118,E1 6.6674,E2 480.5971} C_DIS
LIN {X 112.4091,Y -71.185,Z 177,A -29.9437,B 6.5228,C 0.3151,E1 6.6654,E2 481.9578} C_DIS
LIN {X 110.5759,Y -74.0004,Z 177,A -31.4638,B 6.5226,C 0.3199,E1 6.6631,E2 483.4882} C_DIS
LIN {X 108.7192,Y -76.7021,Z 177,A -32.7308,B 6.5226,C 0.3209,E1 6.6611,E2 484.7388} C_DIS
LIN {X 106.4569,Y -79.8133,Z 177,A -34.387,B 6.5224,C 0.3248,E1 6.6583,E2 486.3965} C_DIS
LIN {X 104.3561,Y -82.5411,Z 177,A -35.9658,B 6.5221,C 0.3298,E1 6.6556,E2 487.9885} C_DIS
LIN {X 101.3029,Y -86.26,Z 177,A -37.8605,B 6.5221,C 0.3316,E1 6.6522,E2 489.8632} C_DIS
LIN {X 99.0937,Y -88.7891,Z 177,A -39.4039,B 6.5218,C 0.3364,E1 6.6493,E2 491.4199} C_DIS
LIN {X 96.3269,Y -91.7836,Z 177,A -41.1351,B 6.5216,C 0.3397,E1 6.646,E2 493.1497} C_DIS
LIN {X 93.47,Y -94.6922,Z 177,A -42.8818,B 6.5214,C 0.3433,E1 6.6426,E2 494.897} C_DIS
LIN {X 90.5133,Y -97.5216,Z 177,A -44.6086,B 6.5213,C 0.3463,E1 6.6391,E2 496.621} C_DIS
LIN {X 86.9404,Y -100.7197,Z 177,A -46.5127,B 6.5212,C 0.3478,E1 6.6351,E2 498.5071} C_DIS
LIN {X 83.8135,Y -103.3368,Z 177,A -48.2302,B 6.521,C 0.3505,E1 6.6314,E2 500.2214} C_DIS
LIN {X 81.1782,Y -105.4199,Z 177,A -49.7911,B 6.5208,C 0.355,E1 6.628,E2 501.7977} C_DIS
LIN {X 77.9387,Y -107.8363,Z 177,A -51.3692,B 6.5208,C 0.3555,E1 6.6244,E2 503.3572} C_DIS
LIN {X 75.2707,Y -109.715,Z 177,A -52.7527,B 6.5206,C 0.3576,E1 6.6213,E2 504.7392} C_DIS
LIN {X 72.477,Y -111.5802,Z 177,A -54.1799,B 6.5206,C 0.3597,E1 6.618,E2 506.1652} C_DIS
LIN {X 69.8011,Y -113.2738,Z 177,A -55.5229,B 6.5204,C 0.3616,E1 6.6148,E2 507.5068} C_DIS
LIN {X 66.9201,Y -114.9994,Z 177,A -57.0924,B 6.5202,C 0.3658,E1 6.611,E2 509.0928} C_DIS
LIN {X 63.1272,Y -117.1241,Z 177,A -58.9152,B 6.5201,C 0.3678,E1 6.6065,E2 510.911} C_DIS
LIN {X 59.7257,Y -118.8944,Z 177,A -60.4476,B 6.5201,C 0.3682,E1 6.6027,E2 512.4299} C_DIS
LIN {X 56.7948,Y -120.3215,Z 177,A -61.8348,B 6.52,C 0.3699,E1 6.5992,E2 513.8162} C_DIS
LIN {X 53.8287,Y -121.6771,Z 177,A -63.2227,B 6.5199,C 0.3714,E1 6.5957,E2 515.2031} C_DIS
LIN {X 50.9055,Y -122.9282,Z 177,A -64.578,B 6.5198,C 0.3728,E1 6.5922,E2 516.5576} C_DIS
LIN {X 47.3079,Y -124.3583,Z 177,A -66.178,B 6.5198,C 0.3737,E1 6.5881,E2 518.1507} C_DIS
LIN {X 44.827,Y -125.2725,Z 177,A -67.3576,B 6.5196,C 0.3756,E1 6.585,E2 519.3361} C_DIS
LIN {X 41.0236,Y -126.57,Z 177,A -69.1586,B 6.5195,C 0.3784,E1 6.5802,E2 521.147} C_DIS
LIN {X 37.0519,Y -127.7883,Z 177,A -70.849,B 6.5195,C 0.3786,E1 6.5757,E2 522.8264} C_DIS
LIN {X 33.8125,Y -128.6839,Z 177,A -72.2848,B 6.5195,C 0.3797,E1 6.5718,E2 524.2618} C_DIS
LIN {X 30.741,Y -129.4519,Z 177,A -73.6458,B 6.5193,C 0.3807,E1 6.5681,E2 525.6234} C_DIS
LIN {X 27.2826,Y -130.2262,Z 177,A -75.1424,B 6.5193,C 0.3814,E1 6.564,E2 527.1174} C_DIS
LIN {X 24.2438,Y -130.8259,Z 177,A -76.4864,B 6.5193,C 0.3824,E1 6.5603,E2 528.4635} C_DIS
LIN {X 21.0324,Y -131.3801,Z 177,A -77.8621,B 6.5193,C 0.3829,E1 6.5566,E2 529.8365} C_DIS
LIN {X 17.9029,Y -131.8427,Z 177,A -79.2526,B 6.5191,C 0.384,E1 6.5527,E2 531.2313} C_DIS
LIN {X 14.6659,Y -132.2413,Z 177,A -80.6517,B 6.5191,C 0.3845,E1 6.5488,E2 532.6305} C_DIS
LIN {X 11.412,Y -132.5612,Z 177,A -82.1245,B 6.5191,C 0.386,E1 6.5447,E2 534.1121} C_DIS
LIN {X 8.0534,Y -132.8075,Z 177,A -83.4709,B 6.5191,C 0.385,E1 6.541,E2 535.4464} C_DIS
LIN {X 4.6346,Y -132.9718,Z 177,A -84.9284,B 6.5191,C 0.3851,E1 6.5369,E2 536.9026} C_DIS
LIN {X 1.632,Y -133.0427,Z 177,A -86.2796,B 6.5191,C 0.3862,E1 6.5331,E2 538.2617} C_DIS
LIN {X 1.632,Y -133.0427,Z 177,A -86.2796,B 6.5191,C 0.3862,E1 6.5331,E2 538.2617} C_DIS
Enddeposition()
LIN {X 0.9684,Y -133.9528,Z 177,A -86.2787,B 6.5194,C 0.3859,E1 6.5335,E2 538.258} C_DIS
Startdeposition()
$VEL.CP = VEL_PRINT
LIN {X 3.6882,Y -133.9055,Z 177,A -84.6063,B 6.5199,C 0.3783,E1 6.5384,E2 536.521} C_DIS
LIN {X 9.0859,Y -133.6493,Z 177,A -82.4409,B 6.5198,C 0.3798,E1 6.5443,E2 534.373} C_DIS
LIN {X 11.7911,Y -133.4372,Z 177,A -81.2136,B 6.5198,C 0.3784,E1 6.5478,E2 533.1366} C_DIS
LIN {X 14.9009,Y -133.126,Z 177,A -79.9448,B 6.5198,C 0.3788,E1 6.5513,E2 531.8757} C_DIS
LIN {X 19.1784,Y -132.5763,Z 177,A -78.0821,B 6.5198,C 0.3776,E1 6.5565,E2 530.0095} C_DIS
LIN {X 23.2568,Y -131.9221,Z 177,A -76.2216,B 6.52,C 0.3752,E1 6.5616,E2 528.1361} C_DIS
LIN {X 27.2509,Y -131.156,Z 177,A -74.6021,B 6.52,C 0.3758,E1 6.566,E2 526.5308} C_DIS
LIN {X 30.559,Y -130.4258,Z 177,A -73.1352,B 6.52,C 0.3745,E1 6.57,E2 525.0608} C_DIS
LIN {X 34.5288,Y -129.4293,Z 177,A -71.3357,B 6.5202,C 0.3722,E1 6.5749,E2 523.2538} C_DIS
LIN {X 38.7697,Y -128.2235,Z 177,A -69.4973,B 6.5202,C 0.3712,E1 6.5798,E2 521.4201} C_DIS
LIN {X 44.515,Y -126.3448,Z 177,A -66.8511,B 6.5205,C 0.3677,E1 6.5869,E2 518.7645} C_DIS
LIN {X 48.5084,Y -124.8642,Z 177,A -64.8246,B 6.5208,C 0.3624,E1 6.5922,E2 516.7106} C_DIS
LIN {X 51.797,Y -123.5364,Z 177,A -63.5904,B 6.5206,C 0.365,E1 6.5953,E2 515.5112} C_DIS
LIN {X 55.1108,Y -122.0948,Z 177,A -62.1796,B 6.5206,C 0.3652,E1 6.5989,E2 514.1162} C_DIS
LIN {X 58.4516,Y -120.5328,Z 177,A -60.5871,B 6.5207,C 0.3628,E1 6.6029,E2 512.5206} C_DIS
LIN {X 61.1408,Y -119.1893,Z 177,A -59.309,B 6.5208,C 0.3611,E1 6.6061,E2 511.2425} C_DIS
LIN {X 64.4715,Y -117.4232,Z 177,A -57.599,B 6.521,C 0.3572,E1 6.6103,E2 509.5189} C_DIS
LIN {X 68.3227,Y -115.2248,Z 177,A -55.7816,B 6.5211,C 0.3556,E1 6.6147,E2 507.71} C_DIS
LIN {X 71.8581,Y -113.0542,Z 177,A -54.1028,B 6.5212,C 0.3543,E1 6.6186,E2 506.0417} C_DIS
LIN {X 74.3398,Y -111.4372,Z 177,A -52.7627,B 6.5214,C 0.351,E1 6.6218,E2 504.6914} C_DIS
LIN {X 77.9084,Y -108.9722,Z 177,A -50.8962,B 6.5216,C 0.3476,E1 6.626,E2 502.8218} C_DIS
LIN {X 81.6067,Y -106.2313,Z 177,A -48.9824,B 6.5217,C 0.3449,E1 6.6303,E2 500.9133} C_DIS
LIN {X 84.8308,Y -103.6745,Z 177,A -47.2538,B 6.5219,C 0.3421,E1 6.634,E2 499.1871} C_DIS
LIN {X 87.8762,Y -101.1063,Z 177,A -45.587,B 6.5219,C 0.3394,E1 6.6376,E2 497.5235} C_DIS
LIN {X 90.9673,Y -98.3351,Z 177,A -43.7602,B 6.5222,C 0.335,E1 6.6414,E2 495.6887} C_DIS
Enddeposition()
END
